KUKA KRL program: EPS_2_251455_MH10A_A_20251003045054.src

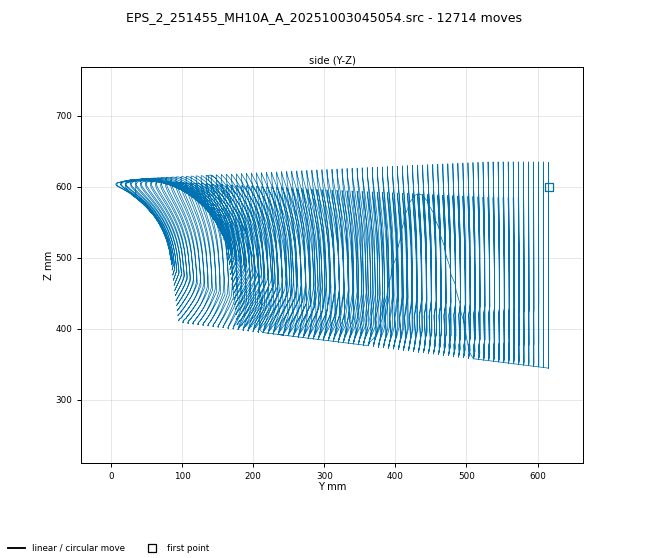
[picture p0: tool path of EPS_2_251455_MH10A_A_20251003045054.src, 12714 of 12716 moves have a stored position in this frame; points joined in program order, loops and branches not executed]
&ACCESS RVP
&REL 4
&COMMENT QRS 19112012
&PARAM EDITMASK = *
DEF PART()
EXT BAS (BAS_COMMAND :IN,REAL :IN )
INT I
BAS (#INITMOV,0 )

;KUKA QRS Post kuka4.cps  Date:22-06-2017 !

File_ID=2866

QRS_PRE_INIT()

;Init var - Until changes are made in qrs_pre_init
Outlet_Square_prg=0
Inlet_1_Square_prg=0
Inlet_2_Square_prg=0
Inlet_3_Square_prg=0
Inlet_4_Square_prg=0
Inlet_5_Square_prg=0

Outlet_1={X 0.000, Y 530.070, Z 534.500, B 0.000, E1 0.000 }
Inlet_1={X 0.000, Y 533.640, Z 484.500, B 0.000, E1 164.000 }
Outlet_1_type=201
Inlet_1_type=201
;QRS#1=Sidecore dimensions
;QRS#2=200-8" PVC SDR 35
;QRS#3=200-8" PVC SDR 35
;QRS#4=
;QRS#5=
;QRS#6=
;QRS#7=
;QRS#8=
;QRS#9=12-08 PSX
;QRS#10=12-08 PSX
;QRS#11=
;QRS#12=
;QRS#13=
;QRS#14=
;QRS#15=
;QRS#16=1220x127x914 3'
;QRS#17=EPS Height
;QRS#18=635
;QRS#19=*
;QRS#20= UPDATED VERSION 22-06-2017
;QRS#21=*
Outlet_Square=0100
Inlet_1_Square=0100
Inlet_2_Square=0
Inlet_3_Square=0
Inlet_4_Square=0
Inlet_5_Square=0
Mill_Square=1
Outlet_Square_Prg=204
Inlet_1_Square_prg=204

QRS_INIT()

$ADVANCE=5

; T1
PTP {E1 173.593,E2 173.593}
PTP {X 0,Y 615.507,A -85,B 0,C 180,E1 173.593,E2 173.593,E3 0,E4 0,E5 0,E6 0}
QRS_SPEED_INIT()
LIN {X 0,Y 615.507,Z 600,A -85,B 0,C 180,E1 173.593,E2 173.593,E3 0,E4 0,E5 0,E6 0} C_VEL
LIN {X 0,Y 615.507,Z 354.862,A -85,B 0,C 180,E1 173.593,E2 173.593} C_VEL
LIN {X 0,Y 615.507,Z 346.684,A -85,B 0,C 180,E1 173.593,E2 173.593} C_VEL
LIN {X 0,Y 615.492,Z 344.684,A -85,B 0,C 180,E1 173.407,E2 173.407} C_VEL
LIN {X 0,Y 615.497,Z 344.7,A -85,B 0,C 180,E1 170.801,E2 170.801} C_VEL
LIN {X 0,Y 615.474,Z 344.687,A -85,B 0,C 180,E1 168.139,E2 168.139} C_VEL
LIN {X 0,Y 615.493,Z 344.685,A -85,B 0,C 180,E1 165.451,E2 165.451} C_VEL
LIN {X 0,Y 615.497,Z 344.694,A -85,B 0,C 180,E1 162.729,E2 162.729} C_VEL
LIN {X 0,Y 615.479,Z 344.684,A -85,B 0,C 180,E1 159.967,E2 159.967} C_VEL
LIN {X 0,Y 615.489,Z 344.696,A -85,B 0,C 180,E1 157.155,E2 157.155} C_VEL
LIN {X 0,Y 615.478,Z 344.686,A -85,B 0,C 180,E1 154.283,E2 154.283} C_VEL
LIN {X 0,Y 615.495,Z 344.686,A -85,B 0,C 180,E1 151.546,E2 151.546} C_VEL
LIN {X 0,Y 615.494,Z 344.695,A -85,B 0,C 180,E1 148.911,E2 148.911} C_VEL
LIN {X 0,Y 615.484,Z 344.686,A -85,B 0,C 180,E1 146.464,E2 146.464} C_VEL
LIN {X 0,Y 615.477,Z 344.685,A -85,B 0,C 180,E1 144.166,E2 144.166} C_VEL
LIN {X 0,Y 615.484,Z 344.684,A -85,B 0,C 180,E1 141.931,E2 141.931} C_VEL
LIN {X 0,Y 615.492,Z 344.695,A -85,B 0,C 180,E1 139.393,E2 139.393} C_VEL
LIN {X 0,Y 615.498,Z 344.685,A -85,B 0,C 180,E1 136.756,E2 136.756} C_VEL
LIN {X 0,Y 615.483,Z 344.685,A -85,B 0,C 180,E1 133.996,E2 133.996} C_VEL
LIN {X 0,Y 615.493,Z 344.693,A -85,B 0,C 180,E1 131.094,E2 131.094} C_VEL
LIN {X 0,Y 615.492,Z 344.688,A -85,B 0,C 180,E1 128.903,E2 128.903} C_VEL
LIN {X 0,Y 615.479,Z 344.684,A -85,B 0,C 180,E1 126.424,E2 126.424} C_VEL
LIN {X 0,Y 615.484,Z 344.851,A -85,B 0,C 180,E1 123.96,E2 123.96} C_VEL
LIN {X 0,Y 615.482,Z 361.283,A -85,B 0,C 180,E1 121.084,E2 121.084} C_VEL
LIN {X 0,Y 615.497,Z 374.419,A -85,B 0,C 180,E1 118.808,E2 118.808} C_VEL
LIN {X 0,Y 615.481,Z 480.795,A -85,B 0,C 180,E1 117.545,E2 117.545} C_VEL
LIN {X 0,Y 615.478,Z 493.507,A -85,B 0,C 180,E1 117.269,E2 117.269} C_VEL
LIN {X 0,Y 615.495,Z 506.255,A -85,B 0,C 180,E1 116.855,E2 116.855} C_VEL
LIN {X 0,Y 615.483,Z 517.741,A -85,B 0,C 180,E1 116.352,E2 116.352} C_VEL
LIN {X 0,Y 615.495,Z 529.018,A -85,B 0,C 180,E1 115.715,E2 115.715} C_VEL
LIN {X 0,Y 615.499,Z 540.401,A -85,B 0,C 180,E1 114.9,E2 114.9} C_VEL
LIN {X 0,Y 615.499,Z 549.036,A -85,B 0,C 180,E1 114.14,E2 114.14} C_VEL
LIN {X 0,Y 615.497,Z 557.732,A -85,B 0,C 180,E1 113.199,E2 113.199} C_VEL
LIN {X 0,Y 615.496,Z 565.632,A -85,B 0,C 180,E1 112.136,E2 112.136} C_VEL
LIN {X 0,Y 615.497,Z 571.832,A -85,B 0,C 180,E1 111.08,E2 111.08} C_VEL
LIN {X 0,Y 615.496,Z 576.587,A -85,B 0,C 180,E1 110.032,E2 110.032} C_VEL
LIN {X 0,Y 615.495,Z 579.049,A -85,B 0,C 180,E1 109.337,E2 109.337} C_VEL
LIN {X 0,Y 615.496,Z 581.148,A -85,B 0,C 180,E1 108.605,E2 108.605} C_VEL
LIN {X 0,Y 615.498,Z 582.545,A -85,B 0,C 180,E1 107.956,E2 107.956} C_VEL
LIN {X 0,Y 615.496,Z 583.573,A -85,B 0,C 180,E1 107.27,E2 107.27} C_VEL
LIN {X 0,Y 615.496,Z 584.282,A -85,B 0,C 180,E1 106.432,E2 106.432} C_VEL
LIN {X 0,Y 615.497,Z 584.12,A -85,B 0,C 180,E1 105.225,E2 105.225} C_VEL
LIN {X 0,Y 615.499,Z 582.513,A -85,B 0,C 180,E1 103.935,E2 103.935} C_VEL
LIN {X 0,Y 615.495,Z 580.869,A -85,B 0,C 180,E1 103.201,E2 103.201} C_VEL
LIN {X 0,Y 615.496,Z 577.77,A -85,B 0,C 180,E1 102.195,E2 102.195} C_VEL
LIN {X 0,Y 615.497,Z 573.606,A -85,B 0,C 180,E1 101.193,E2 101.193} C_VEL
LIN {X 0,Y 615.496,Z 567.248,A -85,B 0,C 180,E1 100.028,E2 100.028} C_VEL
LIN {X 0,Y 615.496,Z 560.341,A -85,B 0,C 180,E1 99.033,E2 99.033} C_VEL
LIN {X 0,Y 615.499,Z 551.708,A -85,B 0,C 180,E1 98.04,E2 98.04} C_VEL
LIN {X 0,Y 615.497,Z 542.889,A -85,B 0,C 180,E1 97.215,E2 97.215} C_VEL
LIN {X 0,Y 615.496,Z 533.241,A -85,B 0,C 180,E1 96.474,E2 96.474} C_VEL
LIN {X 0,Y 615.492,Z 522.644,A -85,B 0,C 180,E1 95.816,E2 95.816} C_VEL
LIN {X 0,Y 615.496,Z 510.844,A -85,B 0,C 180,E1 95.241,E2 95.241} C_VEL
LIN {X 0,Y 615.486,Z 498.624,A -85,B 0,C 180,E1 94.79,E2 94.79} C_VEL
LIN {X 0,Y 615.477,Z 486.033,A -85,B 0,C 180,E1 94.461,E2 94.461} C_VEL
LIN {X 0,Y 615.482,Z 470.995,A -85,B 0,C 180,E1 94.236,E2 94.236} C_VEL
LIN {X 0,Y 615.491,Z 374.345,A -85,B 0,C 180,E1 93.089,E2 93.089} C_VEL
LIN {X 0,Y 615.484,Z 358.413,A -85,B 0,C 180,E1 90.327,E2 90.327} C_VEL
LIN {X 0,Y 615.488,Z 344.686,A -85,B 0,C 180,E1 87.914,E2 87.914} C_VEL
LIN {X 0,Y 615.478,Z 344.685,A -85,B 0,C 180,E1 85.415,E2 85.415} C_VEL
LIN {X 0,Y 615.495,Z 344.693,A -85,B 0,C 180,E1 82.785,E2 82.785} C_VEL
LIN {X 0,Y 615.495,Z 344.687,A -85,B 0,C 180,E1 80.138,E2 80.138} C_VEL
LIN {X 0,Y 615.478,Z 344.685,A -85,B 0,C 180,E1 77.47,E2 77.47} C_VEL
LIN {X 0,Y 615.494,Z 344.696,A -85,B 0,C 180,E1 74.775,E2 74.775} C_VEL
LIN {X 0,Y 615.495,Z 344.683,A -85,B 0,C 180,E1 72.044,E2 72.044} C_VEL
LIN {X 0,Y 615.488,Z 344.686,A -85,B 0,C 180,E1 69.27,E2 69.27} C_VEL
LIN {X 0,Y 615.492,Z 344.692,A -85,B 0,C 180,E1 66.444,E2 66.444} C_VEL
LIN {X 0,Y 615.494,Z 344.687,A -85,B 0,C 180,E1 64.285,E2 64.285} C_VEL
LIN {X 0,Y 615.477,Z 344.686,A -85,B 0,C 180,E1 61.553,E2 61.553} C_VEL
LIN {X 0,Y 615.496,Z 344.697,A -85,B 0,C 180,E1 58.914,E2 58.914} C_VEL
LIN {X 0,Y 615.483,Z 344.683,A -85,B 0,C 180,E1 55.979,E2 55.979} C_VEL
LIN {X 0,Y 615.493,Z 344.695,A -85,B 0,C 180,E1 53.063,E2 53.063} C_VEL
LIN {X 0,Y 615.495,Z 344.683,A -85,B 0,C 180,E1 50.252,E2 50.252} C_VEL
LIN {X 0,Y 615.476,Z 344.687,A -85,B 0,C 180,E1 47.647,E2 47.647} C_VEL
LIN {X 0,Y 615.493,Z 344.7,A -85,B 0,C 180,E1 44.933,E2 44.933} C_VEL
LIN {X 0,Y 615.486,Z 344.683,A -85,B 0,C 180,E1 42.082,E2 42.082} C_VEL
LIN {X 0,Y 615.477,Z 344.686,A -85,B 0,C 180,E1 39.751,E2 39.751} C_VEL
LIN {X 0,Y 615.492,Z 344.697,A -85,B 0,C 180,E1 36.939,E2 36.939} C_VEL
LIN {X 0,Y 615.481,Z 344.684,A -85,B 0,C 180,E1 34.023,E2 34.023} C_VEL
LIN {X 0,Y 615.479,Z 344.688,A -85,B 0,C 180,E1 31.686,E2 31.686} C_VEL
LIN {X 0,Y 615.489,Z 344.693,A -85,B 0,C 180,E1 29.407,E2 29.407} C_VEL
LIN {X 0,Y 615.494,Z 344.682,A -85,B 0,C 180,E1 26.444,E2 26.444} C_VEL
LIN {X 0,Y 615.485,Z 344.692,A -85,B 0,C 180,E1 23.557,E2 23.557} C_VEL
LIN {X 0,Y 615.484,Z 344.688,A -85,B 0,C 180,E1 20.731,E2 20.731} C_VEL
LIN {X 0,Y 615.477,Z 344.687,A -85,B 0,C 180,E1 17.958,E2 17.958} C_VEL
LIN {X 0,Y 615.491,Z 344.699,A -85,B 0,C 180,E1 15.226,E2 15.226} C_VEL
LIN {X 0,Y 615.485,Z 344.683,A -85,B 0,C 180,E1 12.53,E2 12.53} C_VEL
LIN {X 0,Y 615.477,Z 344.69,A -85,B 0,C 180,E1 9.863,E2 9.863} C_VEL
LIN {X 0,Y 615.483,Z 344.697,A -85,B 0,C 180,E1 7.216,E2 7.216} C_VEL
LIN {X 0,Y 615.492,Z 344.682,A -85,B 0,C 180,E1 4.585,E2 4.585} C_VEL
LIN {X 0,Y 615.477,Z 344.69,A -85,B 0,C 180,E1 1.963,E2 1.963} C_VEL
LIN {X 0,Y 615.486,Z 344.698,A -85,B 0,C 180,E1 -0.654,E2 -0.654} C_VEL
LIN {X 0,Y 615.485,Z 344.684,A -85,B 0,C 180,E1 -3.273,E2 -3.273} C_VEL
LIN {X 0,Y 615.476,Z 344.689,A -85,B 0,C 180,E1 -5.899,E2 -5.899} C_VEL
LIN {X 0,Y 615.486,Z 344.699,A -85,B 0,C 180,E1 -8.537,E2 -8.537} C_VEL
LIN {X 0,Y 615.483,Z 344.684,A -85,B 0,C 180,E1 -11.193,E2 -11.193} C_VEL
LIN {X 0,Y 615.48,Z 344.691,A -85,B 0,C 180,E1 -13.935,E2 -13.935} C_VEL
LIN {X 0,Y 615.482,Z 344.695,A -85,B 0,C 180,E1 -16.587,E2 -16.587} C_VEL
LIN {X 0,Y 615.486,Z 344.683,A -85,B 0,C 180,E1 -19.338,E2 -19.338} C_VEL
LIN {X 0,Y 615.488,Z 344.697,A -85,B 0,C 180,E1 -22.136,E2 -22.136} C_VEL
LIN {X 0,Y 615.476,Z 344.686,A -85,B 0,C 180,E1 -24.992,E2 -24.992} C_VEL
LIN {X 0,Y 615.482,Z 344.684,A -85,B 0,C 180,E1 -27.177,E2 -27.177} C_VEL
LIN {X 0,Y 615.483,Z 344.691,A -85,B 0,C 180,E1 -29.796,E2 -29.796} C_VEL
LIN {X 0,Y 615.489,Z 344.692,A -85,B 0,C 180,E1 -32.457,E2 -32.457} C_VEL
LIN {X 0,Y 615.477,Z 344.687,A -85,B 0,C 180,E1 -34.816,E2 -34.816} C_VEL
LIN {X 0,Y 615.489,Z 344.682,A -85,B 0,C 180,E1 -37.242,E2 -37.242} C_VEL
LIN {X 0,Y 615.497,Z 344.7,A -85,B 0,C 180,E1 -40.092,E2 -40.092} C_VEL
LIN {X 0,Y 615.493,Z 344.691,A -85,B 0,C 180,E1 -42.353,E2 -42.353} C_VEL
LIN {X 0,Y 615.481,Z 344.684,A -85,B 0,C 180,E1 -45.069,E2 -45.069} C_VEL
LIN {X 0,Y 615.494,Z 344.699,A -85,B 0,C 180,E1 -47.919,E2 -47.919} C_VEL
LIN {X 0,Y 615.495,Z 344.691,A -85,B 0,C 180,E1 -50.252,E2 -50.252} C_VEL
LIN {X 0,Y 615.483,Z 344.684,A -85,B 0,C 180,E1 -53.064,E2 -53.064} C_VEL
LIN {X 0,Y 615.497,Z 344.698,A -85,B 0,C 180,E1 -55.98,E2 -55.98} C_VEL
LIN {X 0,Y 615.487,Z 344.689,A -85,B 0,C 180,E1 -58.315,E2 -58.315} C_VEL
LIN {X 0,Y 615.477,Z 344.686,A -85,B 0,C 180,E1 -60.594,E2 -60.594} C_VEL
LIN {X 0,Y 615.486,Z 344.683,A -85,B 0,C 180,E1 -62.956,E2 -62.956} C_VEL
LIN {X 0,Y 615.491,Z 344.7,A -85,B 0,C 180,E1 -65.729,E2 -65.729} C_VEL
LIN {X 0,Y 615.487,Z 344.827,A -85,B 0,C 180,E1 -67.067,E2 -67.067} C_VEL
LIN {X 0,Y 615.484,Z 366.758,A -85,B 0,C 180,E1 -69.968,E2 -69.968} C_VEL
LIN {X 0,Y 615.478,Z 388,A -85,B 0,C 180,E1 -72.73,E2 -72.73} C_VEL
LIN {X 0,Y 615.479,Z 409.218,A -85,B 0,C 180,E1 -75.451,E2 -75.451} C_VEL
LIN {X 0,Y 615.497,Z 422.298,A -85,B 0,C 180,E1 -77.114,E2 -77.114} C_VEL
LIN {X 0,Y 615.479,Z 530.847,A -85,B 0,C 180,E1 -78.411,E2 -78.411} C_VEL
LIN {X 0,Y 615.478,Z 543.355,A -85,B 0,C 180,E1 -78.682,E2 -78.682} C_VEL
LIN {X 0,Y 615.491,Z 556.568,A -85,B 0,C 180,E1 -79.111,E2 -79.111} C_VEL
LIN {X 0,Y 615.478,Z 568.483,A -85,B 0,C 180,E1 -79.639,E2 -79.639} C_VEL
LIN {X 0,Y 615.487,Z 579.999,A -85,B 0,C 180,E1 -80.304,E2 -80.304} C_VEL
LIN {X 0,Y 615.499,Z 590.344,A -85,B 0,C 180,E1 -81.05,E2 -81.05} C_VEL
LIN {X 0,Y 615.497,Z 598.814,A -85,B 0,C 180,E1 -81.794,E2 -81.794} C_VEL
LIN {X 0,Y 615.498,Z 606.608,A -85,B 0,C 180,E1 -82.62,E2 -82.62} C_VEL
LIN {X 0,Y 615.496,Z 614.204,A -85,B 0,C 180,E1 -83.608,E2 -83.608} C_VEL
LIN {X 0,Y 615.498,Z 621.205,A -85,B 0,C 180,E1 -84.759,E2 -84.759} C_VEL
LIN {X 0,Y 615.493,Z 625.852,A -85,B 0,C 180,E1 -85.744,E2 -85.744} C_VEL
LIN {X 0,Y 615.495,Z 629.399,A -85,B 0,C 180,E1 -86.727,E2 -86.727} C_VEL
LIN {X 0,Y 615.497,Z 631.233,A -85,B 0,C 180,E1 -87.382,E2 -87.382} C_VEL
LIN {X 0,Y 615.497,Z 632.608,A -85,B 0,C 180,E1 -88.037,E2 -88.037} C_VEL
LIN {X 0,Y 615.496,Z 634.174,A -85,B 0,C 180,E1 -89.346,E2 -89.346} C_VEL
LIN {X 0,Y 615.494,Z 634.389,A -85,B 0,C 180,E1 -90,E2 -90} C_VEL
LIN {X 0,Y 615.496,Z 633.58,A -85,B 0,C 180,E1 -91.309,E2 -91.309} C_VEL
LIN {X 0,Y 615.497,Z 632.608,A -85,B 0,C 180,E1 -91.963,E2 -91.963} C_VEL
LIN {X 0,Y 615.497,Z 631.233,A -85,B 0,C 180,E1 -92.618,E2 -92.618} C_VEL
LIN {X 0,Y 615.496,Z 628.35,A -85,B 0,C 180,E1 -93.601,E2 -93.601} C_VEL
LIN {X 0,Y 615.498,Z 624.442,A -85,B 0,C 180,E1 -94.584,E2 -94.584} C_VEL
LIN {X 0,Y 615.499,Z 619.406,A -85,B 0,C 180,E1 -95.57,E2 -95.57} C_VEL
LIN {X 0,Y 615.497,Z 612.869,A -85,B 0,C 180,E1 -96.583,E2 -96.583} C_VEL
LIN {X 0,Y 615.497,Z 605.135,A -85,B 0,C 180,E1 -97.545,E2 -97.545} C_VEL
LIN {X 0,Y 615.498,Z 597.047,A -85,B 0,C 180,E1 -98.371,E2 -98.371} C_VEL
LIN {X 0,Y 615.499,Z 587.17,A -85,B 0,C 180,E1 -99.198,E2 -99.198} C_VEL
LIN {X 0,Y 615.488,Z 575.985,A -85,B 0,C 180,E1 -99.945,E2 -99.945} C_VEL
LIN {X 0,Y 615.481,Z 565.029,A -85,B 0,C 180,E1 -100.527,E2 -100.527} C_VEL
LIN {X 0,Y 615.49,Z 552.452,A -85,B 0,C 180,E1 -101.041,E2 -101.041} C_VEL
LIN {X 0,Y 615.477,Z 540.079,A -85,B 0,C 180,E1 -101.401,E2 -101.401} C_VEL
LIN {X 0,Y 615.481,Z 526.487,A -85,B 0,C 180,E1 -101.652,E2 -101.652} C_VEL
LIN {X 0,Y 615.497,Z 422.298,A -85,B 0,C 180,E1 -102.886,E2 -102.886} C_VEL
LIN {X 0,Y 615.485,Z 399.937,A -85,B 0,C 180,E1 -105.735,E2 -105.735} C_VEL
LIN {X 0,Y 615.481,Z 377.716,A -85,B 0,C 180,E1 -108.602,E2 -108.602} C_VEL
LIN {X 0,Y 615.478,Z 357.457,A -85,B 0,C 180,E1 -111.256,E2 -111.256} C_VEL
LIN {X 0,Y 615.486,Z 344.684,A -85,B 0,C 180,E1 -112.977,E2 -112.977} C_VEL
LIN {X 0,Y 615.489,Z 344.688,A -85,B 0,C 180,E1 -115.715,E2 -115.715} C_VEL
LIN {X 0,Y 615.49,Z 344.687,A -85,B 0,C 180,E1 -118.657,E2 -118.657} C_VEL
LIN {X 0,Y 615.482,Z 344.684,A -85,B 0,C 180,E1 -121.085,E2 -121.085} C_VEL
LIN {X 0,Y 615.498,Z 344.699,A -85,B 0,C 180,E1 -124.02,E2 -124.02} C_VEL
LIN {X 0,Y 615.483,Z 344.684,A -85,B 0,C 180,E1 -126.936,E2 -126.936} C_VEL
LIN {X 0,Y 615.495,Z 344.692,A -85,B 0,C 180,E1 -129.748,E2 -129.748} C_VEL
LIN {X 0,Y 615.484,Z 344.691,A -85,B 0,C 180,E1 -132.352,E2 -132.352} C_VEL
LIN {X 0,Y 615.479,Z 344.685,A -85,B 0,C 180,E1 -135.068,E2 -135.068} C_VEL
LIN {X 0,Y 615.497,Z 344.7,A -85,B 0,C 180,E1 -137.917,E2 -137.917} C_VEL
LIN {X 0,Y 615.483,Z 344.691,A -85,B 0,C 180,E1 -140.249,E2 -140.249} C_VEL
LIN {X 0,Y 615.478,Z 344.686,A -85,B 0,C 180,E1 -143.063,E2 -143.063} C_VEL
LIN {X 0,Y 615.487,Z 344.696,A -85,B 0,C 180,E1 -145.978,E2 -145.978} C_VEL
LIN {X 0,Y 615.481,Z 344.688,A -85,B 0,C 180,E1 -148.314,E2 -148.314} C_VEL
LIN {X 0,Y 615.487,Z 344.683,A -85,B 0,C 180,E1 -150.594,E2 -150.594} C_VEL
LIN {X 0,Y 615.493,Z 344.697,A -85,B 0,C 180,E1 -153.556,E2 -153.556} C_VEL
LIN {X 0,Y 615.485,Z 344.684,A -85,B 0,C 180,E1 -156.444,E2 -156.444} C_VEL
LIN {X 0,Y 615.48,Z 344.693,A -85,B 0,C 180,E1 -159.269,E2 -159.269} C_VEL
LIN {X 0,Y 615.477,Z 344.69,A -85,B 0,C 180,E1 -162.043,E2 -162.043} C_VEL
LIN {X 0,Y 615.487,Z 344.684,A -85,B 0,C 180,E1 -164.774,E2 -164.774} C_VEL
LIN {X 0,Y 615.488,Z 344.702,A -85,B 0,C 180,E1 -167.47,E2 -167.47} C_VEL
LIN {X 0,Y 615.477,Z 344.687,A -85,B 0,C 180,E1 -170.138,E2 -170.138} C_VEL
LIN {X 0,Y 615.486,Z 344.685,A -85,B 0,C 180,E1 -172.784,E2 -172.784} C_VEL
LIN {X 0,Y 615.5,Z 344.699,A -85,B 0,C 180,E1 -175.416,E2 -175.416} C_VEL
LIN {X 0,Y 615.477,Z 344.687,A -85,B 0,C 180,E1 -178.037,E2 -178.037} C_VEL
LIN {X 0,Y 615.488,Z 344.684,A -85,B 0,C 180,E1 -180.654,E2 -180.654} C_VEL
LIN {X 0,Y 615.493,Z 344.701,A -85,B 0,C 180,E1 -183.273,E2 -183.273} C_VEL
LIN {X 0,Y 615.476,Z 344.688,A -85,B 0,C 180,E1 -185.899,E2 -185.899} C_VEL
LIN {X 0,Y 615.492,Z 344.684,A -85,B 0,C 180,E1 -186.593,E2 -186.593} C_VEL
LIN {X 0,Y 614.818,Z 344.843,A -85,B 0,C 180,E1 -187.139,E2 -187.139} C_VEL
LIN {X 0,Y 611.987,Z 345.247,A -85,B 0,C 180,E1 -188.025,E2 -188.025} C_VEL
LIN {X 0,Y 609.594,Z 345.563,A -85,B 0,C 180,E1 -188.738,E2 -188.738} C_VEL
LIN {X 0,Y 608.554,Z 345.684,A -85,B 0,C 180,E1 -189.287,E2 -189.287} C_VEL
LIN {X 0,Y 608.462,Z 345.692,A -85,B 0,C 180,E1 -189.474,E2 -189.474} C_VEL
LIN {X 0,Y 608.453,Z 345.687,A -85,B 0,C 180,E1 -192,E2 -192} C_VEL
LIN {X 0,Y 608.48,Z 345.688,A -85,B 0,C 180,E1 -194.721,E2 -194.721} C_VEL
LIN {X 0,Y 608.456,Z 345.691,A -85,B 0,C 180,E1 -197.477,E2 -197.477} C_VEL
LIN {X 0,Y 608.461,Z 345.687,A -85,B 0,C 180,E1 -200.275,E2 -200.275} C_VEL
LIN {X 0,Y 608.486,Z 345.685,A -85,B 0,C 180,E1 -202.486,E2 -202.486} C_VEL
LIN {X 0,Y 608.453,Z 345.693,A -85,B 0,C 180,E1 -205.301,E2 -205.301} C_VEL
LIN {X 0,Y 608.449,Z 345.69,A -85,B 0,C 180,E1 -207.518,E2 -207.518} C_VEL
LIN {X 0,Y 608.46,Z 345.686,A -85,B 0,C 180,E1 -209.973,E2 -209.973} C_VEL
LIN {X 0,Y 608.467,Z 345.69,A -85,B 0,C 180,E1 -212.525,E2 -212.525} C_VEL
LIN {X 0,Y 608.444,Z 345.692,A -85,B 0,C 180,E1 -215.278,E2 -215.278} C_VEL
LIN {X 0,Y 608.468,Z 345.685,A -85,B 0,C 180,E1 -217.747,E2 -217.747} C_VEL
LIN {X 0,Y 608.452,Z 345.69,A -85,B 0,C 180,E1 -220.331,E2 -220.331} C_VEL
LIN {X 0,Y 608.484,Z 345.686,A -85,B 0,C 180,E1 -223.312,E2 -223.312} C_VEL
LIN {X 0,Y 608.469,Z 345.687,A -85,B 0,C 180,E1 -226.132,E2 -226.132} C_VEL
LIN {X 0,Y 608.463,Z 345.694,A -85,B 0,C 180,E1 -228.825,E2 -228.825} C_VEL
LIN {X 0,Y 608.471,Z 345.686,A -85,B 0,C 180,E1 -231.413,E2 -231.413} C_VEL
LIN {X 0,Y 608.478,Z 345.686,A -85,B 0,C 180,E1 -233.951,E2 -233.951} C_VEL
LIN {X 0,Y 608.477,Z 345.815,A -85,B 0,C 180,E1 -235.982,E2 -235.982} C_VEL
LIN {X 0,Y 608.478,Z 361.372,A -85,B 0,C 180,E1 -238.729,E2 -238.729} C_VEL
LIN {X 0,Y 608.468,Z 374.62,A -85,B 0,C 180,E1 -241.04,E2 -241.04} C_VEL
LIN {X 0,Y 608.552,Z 481.725,A -85,B 0,C 180,E1 -242.336,E2 -242.336} C_VEL
LIN {X 0,Y 608.522,Z 495.158,A -85,B 0,C 180,E1 -242.643,E2 -242.643} C_VEL
LIN {X 0,Y 608.536,Z 507.968,A -85,B 0,C 180,E1 -243.079,E2 -243.079} C_VEL
LIN {X 0,Y 608.509,Z 519.292,A -85,B 0,C 180,E1 -243.599,E2 -243.599} C_VEL
LIN {X 0,Y 608.5,Z 530.782,A -85,B 0,C 180,E1 -244.275,E2 -244.275} C_VEL
LIN {X 0,Y 608.484,Z 541.548,A -85,B 0,C 180,E1 -245.067,E2 -245.067} C_VEL
LIN {X 0,Y 608.466,Z 550.208,A -85,B 0,C 180,E1 -245.851,E2 -245.851} C_VEL
LIN {X 0,Y 608.471,Z 559.405,A -85,B 0,C 180,E1 -246.877,E2 -246.877} C_VEL
LIN {X 0,Y 608.455,Z 567.1,A -85,B 0,C 180,E1 -247.952,E2 -247.952} C_VEL
LIN {X 0,Y 608.434,Z 573.088,A -85,B 0,C 180,E1 -249.018,E2 -249.018} C_VEL
LIN {X 0,Y 608.435,Z 577.702,A -85,B 0,C 180,E1 -250.078,E2 -250.078} C_VEL
LIN {X 0,Y 608.43,Z 581.545,A -85,B 0,C 180,E1 -251.297,E2 -251.297} C_VEL
LIN {X 0,Y 608.421,Z 583.95,A -85,B 0,C 180,E1 -252.523,E2 -252.523} C_VEL
LIN {X 0,Y 608.423,Z 584.856,A -85,B 0,C 180,E1 -253.487,E2 -253.487} C_VEL
LIN {X 0,Y 608.42,Z 584.862,A -85,B 0,C 180,E1 -254.593,E2 -254.593} C_VEL
LIN {X 0,Y 608.418,Z 584.29,A -85,B 0,C 180,E1 -255.278,E2 -255.278} C_VEL
LIN {X 0,Y 608.446,Z 583.262,A -85,B 0,C 180,E1 -255.994,E2 -255.994} C_VEL
LIN {X 0,Y 608.438,Z 581.93,A -85,B 0,C 180,E1 -256.643,E2 -256.643} C_VEL
LIN {X 0,Y 608.433,Z 578.981,A -85,B 0,C 180,E1 -257.661,E2 -257.661} C_VEL
LIN {X 0,Y 608.43,Z 574.981,A -85,B 0,C 180,E1 -258.676,E2 -258.676} C_VEL
LIN {X 0,Y 608.444,Z 568.822,A -85,B 0,C 180,E1 -259.855,E2 -259.855} C_VEL
LIN {X 0,Y 608.47,Z 562.103,A -85,B 0,C 180,E1 -260.862,E2 -260.862} C_VEL
LIN {X 0,Y 608.464,Z 553.803,A -85,B 0,C 180,E1 -261.866,E2 -261.866} C_VEL
LIN {X 0,Y 608.478,Z 545.303,A -85,B 0,C 180,E1 -262.701,E2 -262.701} C_VEL
LIN {X 0,Y 608.481,Z 534.872,A -85,B 0,C 180,E1 -263.534,E2 -263.534} C_VEL
LIN {X 0,Y 608.513,Z 524.576,A -85,B 0,C 180,E1 -264.2,E2 -264.2} C_VEL
LIN {X 0,Y 608.53,Z 513.328,A -85,B 0,C 180,E1 -264.782,E2 -264.782} C_VEL
LIN {X 0,Y 608.527,Z 501.849,A -85,B 0,C 180,E1 -265.239,E2 -265.239} C_VEL
LIN {X 0,Y 608.539,Z 488.732,A -85,B 0,C 180,E1 -265.612,E2 -265.612} C_VEL
LIN {X 0,Y 608.544,Z 476.006,A -85,B 0,C 180,E1 -265.84,E2 -265.84} C_VEL
LIN {X 0,Y 608.485,Z 374.794,A -85,B 0,C 180,E1 -267.041,E2 -267.041} C_VEL
LIN {X 0,Y 608.46,Z 359.621,A -85,B 0,C 180,E1 -269.669,E2 -269.669} C_VEL
LIN {X 0,Y 608.466,Z 345.688,A -85,B 0,C 180,E1 -272.151,E2 -272.151} C_VEL
LIN {X 0,Y 608.448,Z 345.688,A -85,B 0,C 180,E1 -274.638,E2 -274.638} C_VEL
LIN {X 0,Y 608.472,Z 345.693,A -85,B 0,C 180,E1 -277.299,E2 -277.299} C_VEL
LIN {X 0,Y 608.462,Z 345.688,A -85,B 0,C 180,E1 -279.977,E2 -279.977} C_VEL
LIN {X 0,Y 608.472,Z 345.686,A -85,B 0,C 180,E1 -282.677,E2 -282.677} C_VEL
LIN {X 0,Y 608.478,Z 345.694,A -85,B 0,C 180,E1 -285.405,E2 -285.405} C_VEL
LIN {X 0,Y 608.454,Z 345.687,A -85,B 0,C 180,E1 -288.171,E2 -288.171} C_VEL
LIN {X 0,Y 608.46,Z 345.692,A -85,B 0,C 180,E1 -290.981,E2 -290.981} C_VEL
LIN {X 0,Y 608.469,Z 345.687,A -85,B 0,C 180,E1 -293.844,E2 -293.844} C_VEL
LIN {X 0,Y 608.447,Z 345.688,A -85,B 0,C 180,E1 -296.035,E2 -296.035} C_VEL
LIN {X 0,Y 608.47,Z 345.687,A -85,B 0,C 180,E1 -298.618,E2 -298.618} C_VEL
LIN {X 0,Y 608.481,Z 345.692,A -85,B 0,C 180,E1 -301.315,E2 -301.315} C_VEL
LIN {X 0,Y 608.474,Z 345.686,A -85,B 0,C 180,E1 -303.734,E2 -303.734} C_VEL
LIN {X 0,Y 608.476,Z 345.684,A -85,B 0,C 180,E1 -306.089,E2 -306.089} C_VEL
LIN {X 0,Y 608.473,Z 345.687,A -85,B 0,C 180,E1 -308.587,E2 -308.587} C_VEL
LIN {X 0,Y 608.464,Z 345.692,A -85,B 0,C 180,E1 -311.342,E2 -311.342} C_VEL
LIN {X 0,Y 608.45,Z 345.688,A -85,B 0,C 180,E1 -314.263,E2 -314.263} C_VEL
LIN {X 0,Y 608.462,Z 345.697,A -85,B 0,C 180,E1 -317.04,E2 -317.04} C_VEL
LIN {X 0,Y 608.453,Z 345.688,A -85,B 0,C 180,E1 -319.696,E2 -319.696} C_VEL
LIN {X 0,Y 608.469,Z 345.686,A -85,B 0,C 180,E1 -322.253,E2 -322.253} C_VEL
LIN {X 0,Y 608.474,Z 345.692,A -85,B 0,C 180,E1 -325.089,E2 -325.089} C_VEL
LIN {X 0,Y 608.469,Z 345.685,A -85,B 0,C 180,E1 -327.905,E2 -327.905} C_VEL
LIN {X 0,Y 608.462,Z 345.688,A -85,B 0,C 180,E1 -330.22,E2 -330.22} C_VEL
LIN {X 0,Y 608.482,Z 345.694,A -85,B 0,C 180,E1 -332.789,E2 -332.789} C_VEL
LIN {X 0,Y 608.454,Z 345.689,A -85,B 0,C 180,E1 -335.429,E2 -335.429} C_VEL
LIN {X 0,Y 608.471,Z 345.688,A -85,B 0,C 180,E1 -338.308,E2 -338.308} C_VEL
LIN {X 0,Y 608.467,Z 345.688,A -85,B 0,C 180,E1 -341.281,E2 -341.281} C_VEL
LIN {X 0,Y 608.456,Z 345.687,A -85,B 0,C 180,E1 -343.906,E2 -343.906} C_VEL
LIN {X 0,Y 608.465,Z 345.696,A -85,B 0,C 180,E1 -346.643,E2 -346.643} C_VEL
LIN {X 0,Y 608.466,Z 345.686,A -85,B 0,C 180,E1 -349.35,E2 -349.35} C_VEL
LIN {X 0,Y 608.47,Z 345.687,A -85,B 0,C 180,E1 -352.033,E2 -352.033} C_VEL
LIN {X 0,Y 608.465,Z 345.694,A -85,B 0,C 180,E1 -354.698,E2 -354.698} C_VEL
LIN {X 0,Y 608.479,Z 345.684,A -85,B 0,C 180,E1 -357.352,E2 -357.352} C_VEL
LIN {X 0,Y 608.468,Z 345.688,A -85,B 0,C 180,E1 -360,E2 -360} C_VEL
LIN {X 0,Y 608.48,Z 345.692,A -85,B 0,C 180,E1 -362.648,E2 -362.648} C_VEL
LIN {X 0,Y 608.462,Z 345.686,A -85,B 0,C 180,E1 -365.302,E2 -365.302} C_VEL
LIN {X 0,Y 608.47,Z 345.688,A -85,B 0,C 180,E1 -367.967,E2 -367.967} C_VEL
LIN {X 0,Y 608.465,Z 345.692,A -85,B 0,C 180,E1 -370.65,E2 -370.65} C_VEL
LIN {X 0,Y 608.46,Z 345.686,A -85,B 0,C 180,E1 -373.356,E2 -373.356} C_VEL
LIN {X 0,Y 608.458,Z 345.693,A -85,B 0,C 180,E1 -376.094,E2 -376.094} C_VEL
LIN {X 0,Y 608.45,Z 345.69,A -85,B 0,C 180,E1 -378.87,E2 -378.87} C_VEL
LIN {X 0,Y 608.473,Z 345.687,A -85,B 0,C 180,E1 -381.691,E2 -381.691} C_VEL
LIN {X 0,Y 608.451,Z 345.693,A -85,B 0,C 180,E1 -384.571,E2 -384.571} C_VEL
LIN {X 0,Y 608.473,Z 345.685,A -85,B 0,C 180,E1 -387.209,E2 -387.209} C_VEL
LIN {X 0,Y 608.468,Z 345.692,A -85,B 0,C 180,E1 -389.974,E2 -389.974} C_VEL
LIN {X 0,Y 608.462,Z 345.691,A -85,B 0,C 180,E1 -392.525,E2 -392.525} C_VEL
LIN {X 0,Y 608.439,Z 345.689,A -85,B 0,C 180,E1 -395.278,E2 -395.278} C_VEL
LIN {X 0,Y 608.472,Z 345.689,A -85,B 0,C 180,E1 -397.746,E2 -397.746} C_VEL
LIN {X 0,Y 608.476,Z 345.69,A -85,B 0,C 180,E1 -400.333,E2 -400.333} C_VEL
LIN {X 0,Y 608.483,Z 345.684,A -85,B 0,C 180,E1 -403.312,E2 -403.312} C_VEL
LIN {X 0,Y 608.472,Z 345.693,A -85,B 0,C 180,E1 -406.132,E2 -406.132} C_VEL
LIN {X 0,Y 608.45,Z 345.688,A -85,B 0,C 180,E1 -408.824,E2 -408.824} C_VEL
LIN {X 0,Y 608.471,Z 345.687,A -85,B 0,C 180,E1 -411.413,E2 -411.413} C_VEL
LIN {X 0,Y 608.478,Z 345.695,A -85,B 0,C 180,E1 -413.951,E2 -413.951} C_VEL
LIN {X 0,Y 608.464,Z 345.689,A -85,B 0,C 180,E1 -416.33,E2 -416.33} C_VEL
LIN {X 0,Y 608.476,Z 345.685,A -85,B 0,C 180,E1 -418.728,E2 -418.728} C_VEL
LIN {X 0,Y 608.477,Z 345.688,A -85,B 0,C 180,E1 -421.38,E2 -421.38} C_VEL
LIN {X 0,Y 608.471,Z 345.688,A -85,B 0,C 180,E1 -424.28,E2 -424.28} C_VEL
LIN {X 0,Y 608.479,Z 345.824,A -85,B 0,C 180,E1 -426.923,E2 -426.923} C_VEL
LIN {X 0,Y 608.582,Z 361.447,A -85,B 0,C 180,E1 -429.024,E2 -429.024} C_VEL
LIN {X 0,Y 608.518,Z 382.72,A -85,B 0,C 180,E1 -431.831,E2 -431.831} C_VEL
LIN {X 0,Y 608.492,Z 402.663,A -85,B 0,C 180,E1 -434.423,E2 -434.423} C_VEL
LIN {X 0,Y 608.503,Z 422.524,A -85,B 0,C 180,E1 -436.974,E2 -436.974} C_VEL
LIN {X 0,Y 608.538,Z 530.962,A -85,B 0,C 180,E1 -438.277,E2 -438.277} C_VEL
LIN {X 0,Y 608.514,Z 544.226,A -85,B 0,C 180,E1 -438.572,E2 -438.572} C_VEL
LIN {X 0,Y 608.517,Z 556.598,A -85,B 0,C 180,E1 -438.981,E2 -438.981} C_VEL
LIN {X 0,Y 608.498,Z 568.639,A -85,B 0,C 180,E1 -439.519,E2 -439.519} C_VEL
LIN {X 0,Y 608.48,Z 580.201,A -85,B 0,C 180,E1 -440.191,E2 -440.191} C_VEL
LIN {X 0,Y 608.485,Z 590.596,A -85,B 0,C 180,E1 -440.946,E2 -440.946} C_VEL
LIN {X 0,Y 608.475,Z 599.114,A -85,B 0,C 180,E1 -441.699,E2 -441.699} C_VEL
LIN {X 0,Y 608.471,Z 606.962,A -85,B 0,C 180,E1 -442.534,E2 -442.534} C_VEL
LIN {X 0,Y 608.46,Z 614.287,A -85,B 0,C 180,E1 -443.485,E2 -443.485} C_VEL
LIN {X 0,Y 608.45,Z 619.867,A -85,B 0,C 180,E1 -444.366,E2 -444.366} C_VEL
LIN {X 0,Y 608.432,Z 624.951,A -85,B 0,C 180,E1 -445.362,E2 -445.362} C_VEL
LIN {X 0,Y 608.449,Z 628.896,A -85,B 0,C 180,E1 -446.358,E2 -446.358} C_VEL
LIN {X 0,Y 608.425,Z 631.809,A -85,B 0,C 180,E1 -447.352,E2 -447.352} C_VEL
LIN {X 0,Y 608.442,Z 633.201,A -85,B 0,C 180,E1 -448.014,E2 -448.014} C_VEL
LIN {X 0,Y 608.438,Z 634.783,A -85,B 0,C 180,E1 -449.338,E2 -449.338} C_VEL
LIN {X 0,Y 608.434,Z 635,A -85,B 0,C 180,E1 -450,E2 -450} C_VEL
LIN {X 0,Y 608.448,Z 634.184,A -85,B 0,C 180,E1 -451.324,E2 -451.324} C_VEL
LIN {X 0,Y 608.442,Z 633.201,A -85,B 0,C 180,E1 -451.986,E2 -451.986} C_VEL
LIN {X 0,Y 608.425,Z 631.809,A -85,B 0,C 180,E1 -452.648,E2 -452.648} C_VEL
LIN {X 0,Y 608.449,Z 628.896,A -85,B 0,C 180,E1 -453.642,E2 -453.642} C_VEL
LIN {X 0,Y 608.432,Z 624.95,A -85,B 0,C 180,E1 -454.638,E2 -454.638} C_VEL
LIN {X 0,Y 608.437,Z 618.877,A -85,B 0,C 180,E1 -455.801,E2 -455.801} C_VEL
LIN {X 0,Y 608.462,Z 612.236,A -85,B 0,C 180,E1 -456.799,E2 -456.799} C_VEL
LIN {X 0,Y 608.455,Z 603.991,A -85,B 0,C 180,E1 -457.8,E2 -457.8} C_VEL
LIN {X 0,Y 608.472,Z 595.538,A -85,B 0,C 180,E1 -458.636,E2 -458.636} C_VEL
LIN {X 0,Y 608.471,Z 585.094,A -85,B 0,C 180,E1 -459.473,E2 -459.473} C_VEL
LIN {X 0,Y 608.494,Z 574.76,A -85,B 0,C 180,E1 -460.144,E2 -460.144} C_VEL
LIN {X 0,Y 608.521,Z 563.255,A -85,B 0,C 180,E1 -460.74,E2 -460.74} C_VEL
LIN {X 0,Y 608.531,Z 550.887,A -85,B 0,C 180,E1 -461.225,E2 -461.225} C_VEL
LIN {X 0,Y 608.537,Z 537.45,A -85,B 0,C 180,E1 -461.597,E2 -461.597} C_VEL
LIN {X 0,Y 608.546,Z 525.105,A -85,B 0,C 180,E1 -461.808,E2 -461.808} C_VEL
LIN {X 0,Y 608.493,Z 422.441,A -85,B 0,C 180,E1 -463.037,E2 -463.037} C_VEL
LIN {X 0,Y 608.494,Z 400.004,A -85,B 0,C 180,E1 -465.92,E2 -465.92} C_VEL
LIN {X 0,Y 608.54,Z 378.405,A -85,B 0,C 180,E1 -468.735,E2 -468.735} C_VEL
LIN {X 0,Y 608.563,Z 357.458,A -85,B 0,C 180,E1 -471.51,E2 -471.51} C_VEL
LIN {X 0,Y 608.468,Z 345.687,A -85,B 0,C 180,E1 -473.1,E2 -473.1} C_VEL
LIN {X 0,Y 608.471,Z 345.688,A -85,B 0,C 180,E1 -475.72,E2 -475.72} C_VEL
LIN {X 0,Y 608.476,Z 345.688,A -85,B 0,C 180,E1 -478.62,E2 -478.62} C_VEL
LIN {X 0,Y 608.475,Z 345.685,A -85,B 0,C 180,E1 -481.315,E2 -481.315} C_VEL
LIN {X 0,Y 608.473,Z 345.69,A -85,B 0,C 180,E1 -483.735,E2 -483.735} C_VEL
LIN {X 0,Y 608.477,Z 345.695,A -85,B 0,C 180,E1 -486.089,E2 -486.089} C_VEL
LIN {X 0,Y 608.471,Z 345.687,A -85,B 0,C 180,E1 -488.587,E2 -488.587} C_VEL
LIN {X 0,Y 608.457,Z 345.688,A -85,B 0,C 180,E1 -491.341,E2 -491.341} C_VEL
LIN {X 0,Y 608.457,Z 345.692,A -85,B 0,C 180,E1 -494.264,E2 -494.264} C_VEL
LIN {X 0,Y 608.453,Z 345.687,A -85,B 0,C 180,E1 -497.04,E2 -497.04} C_VEL
LIN {X 0,Y 608.455,Z 345.695,A -85,B 0,C 180,E1 -499.697,E2 -499.697} C_VEL
LIN {X 0,Y 608.471,Z 345.689,A -85,B 0,C 180,E1 -502.254,E2 -502.254} C_VEL
LIN {X 0,Y 608.469,Z 345.686,A -85,B 0,C 180,E1 -505.09,E2 -505.09} C_VEL
LIN {X 0,Y 608.47,Z 345.693,A -85,B 0,C 180,E1 -507.906,E2 -507.906} C_VEL
LIN {X 0,Y 608.464,Z 345.689,A -85,B 0,C 180,E1 -510.22,E2 -510.22} C_VEL
LIN {X 0,Y 608.475,Z 345.685,A -85,B 0,C 180,E1 -512.791,E2 -512.791} C_VEL
LIN {X 0,Y 608.449,Z 345.694,A -85,B 0,C 180,E1 -515.429,E2 -515.429} C_VEL
LIN {X 0,Y 608.471,Z 345.686,A -85,B 0,C 180,E1 -518.309,E2 -518.309} C_VEL
LIN {X 0,Y 608.466,Z 345.691,A -85,B 0,C 180,E1 -521.281,E2 -521.281} C_VEL
LIN {X 0,Y 608.456,Z 345.691,A -85,B 0,C 180,E1 -523.906,E2 -523.906} C_VEL
LIN {X 0,Y 608.46,Z 345.686,A -85,B 0,C 180,E1 -526.644,E2 -526.644} C_VEL
LIN {X 0,Y 608.466,Z 345.694,A -85,B 0,C 180,E1 -529.35,E2 -529.35} C_VEL
LIN {X 0,Y 608.47,Z 345.687,A -85,B 0,C 180,E1 -532.033,E2 -532.033} C_VEL
LIN {X 0,Y 608.464,Z 345.687,A -85,B 0,C 180,E1 -534.698,E2 -534.698} C_VEL
LIN {X 0,Y 608.484,Z 345.694,A -85,B 0,C 180,E1 -537.352,E2 -537.352} C_VEL
LIN {X 0,Y 608.468,Z 345.687,A -85,B 0,C 180,E1 -540,E2 -540} C_VEL
LIN {X 0,Y 608.482,Z 345.685,A -85,B 0,C 180,E1 -542.648,E2 -542.648} C_VEL
LIN {X 0,Y 608.473,Z 345.695,A -85,B 0,C 180,E1 -545.302,E2 -545.302} C_VEL
LIN {X 0,Y 608.47,Z 345.686,A -85,B 0,C 180,E1 -547.967,E2 -547.967} C_VEL
LIN {X 0,Y 608.462,Z 345.692,A -85,B 0,C 180,E1 -549.474,E2 -549.474} C_VEL
LIN {X 0,Y 607.774,Z 345.774,A -85,B 0,C 180,E1 -550.026,E2 -550.026} C_VEL
LIN {X 0,Y 604.913,Z 346.134,A -85,B 0,C 180,E1 -550.923,E2 -550.923} C_VEL
LIN {X 0,Y 602.511,Z 346.43,A -85,B 0,C 180,E1 -551.645,E2 -551.645} C_VEL
LIN {X 0,Y 601.487,Z 346.555,A -85,B 0,C 180,E1 -552.201,E2 -552.201} C_VEL
LIN {X 0,Y 601.406,Z 346.565,A -85,B 0,C 180,E1 -552.39,E2 -552.39} C_VEL
LIN {X 0,Y 601.433,Z 346.568,A -85,B 0,C 180,E1 -554.897,E2 -554.897} C_VEL
LIN {X 0,Y 601.398,Z 346.568,A -85,B 0,C 180,E1 -557.689,E2 -557.689} C_VEL
LIN {X 0,Y 601.431,Z 346.564,A -85,B 0,C 180,E1 -560.522,E2 -560.522} C_VEL
LIN {X 0,Y 601.418,Z 346.568,A -85,B 0,C 180,E1 -563.411,E2 -563.411} C_VEL
LIN {X 0,Y 601.406,Z 346.567,A -85,B 0,C 180,E1 -566.364,E2 -566.364} C_VEL
LIN {X 0,Y 601.442,Z 346.569,A -85,B 0,C 180,E1 -568.792,E2 -568.792} C_VEL
LIN {X 0,Y 601.413,Z 346.565,A -85,B 0,C 180,E1 -571.727,E2 -571.727} C_VEL
LIN {X 0,Y 601.428,Z 346.563,A -85,B 0,C 180,E1 -574.119,E2 -574.119} C_VEL
LIN {X 0,Y 601.413,Z 346.57,A -85,B 0,C 180,E1 -576.583,E2 -576.583} C_VEL
LIN {X 0,Y 601.436,Z 346.562,A -85,B 0,C 180,E1 -579.537,E2 -579.537} C_VEL
LIN {X 0,Y 601.438,Z 346.569,A -85,B 0,C 180,E1 -582.595,E2 -582.595} C_VEL
LIN {X 0,Y 601.423,Z 346.564,A -85,B 0,C 180,E1 -585.483,E2 -585.483} C_VEL
LIN {X 0,Y 601.427,Z 346.568,A -85,B 0,C 180,E1 -588.407,E2 -588.407} C_VEL
LIN {X 0,Y 601.439,Z 346.568,A -85,B 0,C 180,E1 -590.877,E2 -590.877} C_VEL
LIN {X 0,Y 601.444,Z 346.561,A -85,B 0,C 180,E1 -593.735,E2 -593.735} C_VEL
LIN {X 0,Y 601.42,Z 346.646,A -85,B 0,C 180,E1 -595.912,E2 -595.912} C_VEL
LIN {X 0,Y 601.443,Z 361.359,A -85,B 0,C 180,E1 -598.543,E2 -598.543} C_VEL
LIN {X 0,Y 601.412,Z 374.66,A -85,B 0,C 180,E1 -600.891,E2 -600.891} C_VEL
LIN {X 0,Y 601.684,Z 380.406,A -85,B 0,C 180,E1 -600.966,E2 -600.966} C_VEL
LIN {X 0,Y 601.594,Z 481.501,A -85,B 0,C 180,E1 -602.195,E2 -602.195} C_VEL
LIN {X 0,Y 601.551,Z 495.079,A -85,B 0,C 180,E1 -602.507,E2 -602.507} C_VEL
LIN {X 0,Y 601.564,Z 507.771,A -85,B 0,C 180,E1 -602.942,E2 -602.942} C_VEL
LIN {X 0,Y 601.499,Z 518.891,A -85,B 0,C 180,E1 -603.455,E2 -603.455} C_VEL
LIN {X 0,Y 601.465,Z 530.246,A -85,B 0,C 180,E1 -604.124,E2 -604.124} C_VEL
LIN {X 0,Y 601.465,Z 541.295,A -85,B 0,C 180,E1 -604.94,E2 -604.94} C_VEL
LIN {X 0,Y 601.4,Z 551.203,A -85,B 0,C 180,E1 -605.858,E2 -605.858} C_VEL
LIN {X 0,Y 601.386,Z 559.233,A -85,B 0,C 180,E1 -606.771,E2 -606.771} C_VEL
LIN {X 0,Y 601.392,Z 566.085,A -85,B 0,C 180,E1 -607.723,E2 -607.723} C_VEL
LIN {X 0,Y 601.344,Z 572.104,A -85,B 0,C 180,E1 -608.759,E2 -608.759} C_VEL
LIN {X 0,Y 601.342,Z 576.969,A -85,B 0,C 180,E1 -609.833,E2 -609.833} C_VEL
LIN {X 0,Y 601.332,Z 580.578,A -85,B 0,C 180,E1 -610.899,E2 -610.899} C_VEL
LIN {X 0,Y 601.325,Z 582.338,A -85,B 0,C 180,E1 -611.606,E2 -611.606} C_VEL
LIN {X 0,Y 601.314,Z 583.652,A -85,B 0,C 180,E1 -612.31,E2 -612.31} C_VEL
LIN {X 0,Y 601.322,Z 584.81,A -85,B 0,C 180,E1 -613.414,E2 -613.414} C_VEL
LIN {X 0,Y 601.327,Z 584.922,A -85,B 0,C 180,E1 -614.407,E2 -614.407} C_VEL
LIN {X 0,Y 601.315,Z 584.508,A -85,B 0,C 180,E1 -615.101,E2 -615.101} C_VEL
LIN {X 0,Y 601.353,Z 583.395,A -85,B 0,C 180,E1 -615.937,E2 -615.937} C_VEL
LIN {X 0,Y 601.328,Z 580.634,A -85,B 0,C 180,E1 -617.17,E2 -617.17} C_VEL
LIN {X 0,Y 601.351,Z 577.188,A -85,B 0,C 180,E1 -618.199,E2 -618.199} C_VEL
LIN {X 0,Y 601.34,Z 572.649,A -85,B 0,C 180,E1 -619.223,E2 -619.223} C_VEL
LIN {X 0,Y 601.377,Z 565.774,A -85,B 0,C 180,E1 -620.414,E2 -620.414} C_VEL
LIN {X 0,Y 601.407,Z 558.324,A -85,B 0,C 180,E1 -621.431,E2 -621.431} C_VEL
LIN {X 0,Y 601.397,Z 550.774,A -85,B 0,C 180,E1 -622.277,E2 -622.277} C_VEL
LIN {X 0,Y 601.452,Z 541.647,A -85,B 0,C 180,E1 -623.121,E2 -623.121} C_VEL
LIN {X 0,Y 601.485,Z 530.28,A -85,B 0,C 180,E1 -623.964,E2 -623.964} C_VEL
LIN {X 0,Y 601.5,Z 518.868,A -85,B 0,C 180,E1 -624.637,E2 -624.637} C_VEL
LIN {X 0,Y 601.573,Z 506.846,A -85,B 0,C 180,E1 -625.183,E2 -625.183} C_VEL
LIN {X 0,Y 601.554,Z 493.636,A -85,B 0,C 180,E1 -625.624,E2 -625.624} C_VEL
LIN {X 0,Y 601.591,Z 480.258,A -85,B 0,C 180,E1 -625.918,E2 -625.918} C_VEL
LIN {X 0,Y 601.542,Z 375.529,A -85,B 0,C 180,E1 -627.185,E2 -627.185} C_VEL
LIN {X 0,Y 601.413,Z 374.442,A -85,B 0,C 180,E1 -627.237,E2 -627.237} C_VEL
LIN {X 0,Y 601.451,Z 358.811,A -85,B 0,C 180,E1 -630,E2 -630} C_VEL
LIN {X 0,Y 601.424,Z 346.566,A -85,B 0,C 180,E1 -632.218,E2 -632.218} C_VEL
LIN {X 0,Y 601.419,Z 346.564,A -85,B 0,C 180,E1 -634.692,E2 -634.692} C_VEL
LIN {X 0,Y 601.449,Z 346.57,A -85,B 0,C 180,E1 -637.385,E2 -637.385} C_VEL
LIN {X 0,Y 601.438,Z 346.562,A -85,B 0,C 180,E1 -640.095,E2 -640.095} C_VEL
LIN {X 0,Y 601.42,Z 346.565,A -85,B 0,C 180,E1 -642.828,E2 -642.828} C_VEL
LIN {X 0,Y 601.419,Z 346.57,A -85,B 0,C 180,E1 -645.591,E2 -645.591} C_VEL
LIN {X 0,Y 601.424,Z 346.563,A -85,B 0,C 180,E1 -648.391,E2 -648.391} C_VEL
LIN {X 0,Y 601.412,Z 346.574,A -85,B 0,C 180,E1 -651.239,E2 -651.239} C_VEL
LIN {X 0,Y 601.456,Z 346.559,A -85,B 0,C 180,E1 -654.14,E2 -654.14} C_VEL
LIN {X 0,Y 601.455,Z 346.568,A -85,B 0,C 180,E1 -657.11,E2 -657.11} C_VEL
LIN {X 0,Y 601.426,Z 346.57,A -85,B 0,C 180,E1 -659.392,E2 -659.392} C_VEL
LIN {X 0,Y 601.414,Z 346.566,A -85,B 0,C 180,E1 -661.725,E2 -661.725} C_VEL
LIN {X 0,Y 601.431,Z 346.562,A -85,B 0,C 180,E1 -664.117,E2 -664.117} C_VEL
LIN {X 0,Y 601.416,Z 346.566,A -85,B 0,C 180,E1 -666.581,E2 -666.581} C_VEL
LIN {X 0,Y 601.445,Z 346.564,A -85,B 0,C 180,E1 -669.535,E2 -669.535} C_VEL
LIN {X 0,Y 601.409,Z 346.568,A -85,B 0,C 180,E1 -672.59,E2 -672.59} C_VEL
LIN {X 0,Y 601.422,Z 346.566,A -85,B 0,C 180,E1 -674.534,E2 -674.534} C_VEL
LIN {X 0,Y 601.438,Z 346.565,A -85,B 0,C 180,E1 -677.405,E2 -677.405} C_VEL
LIN {X 0,Y 601.437,Z 346.564,A -85,B 0,C 180,E1 -680.463,E2 -680.463} C_VEL
LIN {X 0,Y 601.414,Z 346.567,A -85,B 0,C 180,E1 -683.417,E2 -683.417} C_VEL
LIN {X 0,Y 601.428,Z 346.563,A -85,B 0,C 180,E1 -686.063,E2 -686.063} C_VEL
LIN {X 0,Y 601.438,Z 346.566,A -85,B 0,C 180,E1 -688.54,E2 -688.54} C_VEL
LIN {X 0,Y 601.434,Z 346.564,A -85,B 0,C 180,E1 -691.373,E2 -691.373} C_VEL
LIN {X 0,Y 601.405,Z 346.566,A -85,B 0,C 180,E1 -693.636,E2 -693.636} C_VEL
LIN {X 0,Y 601.416,Z 346.571,A -85,B 0,C 180,E1 -696.589,E2 -696.589} C_VEL
LIN {X 0,Y 601.429,Z 346.563,A -85,B 0,C 180,E1 -699.478,E2 -699.478} C_VEL
LIN {X 0,Y 601.398,Z 346.57,A -85,B 0,C 180,E1 -702.311,E2 -702.311} C_VEL
LIN {X 0,Y 601.414,Z 346.57,A -85,B 0,C 180,E1 -704.408,E2 -704.408} C_VEL
LIN {X 0,Y 601.421,Z 346.566,A -85,B 0,C 180,E1 -707.172,E2 -707.172} C_VEL
LIN {X 0,Y 601.428,Z 346.563,A -85,B 0,C 180,E1 -709.905,E2 -709.905} C_VEL
LIN {X 0,Y 601.445,Z 346.571,A -85,B 0,C 180,E1 -712.615,E2 -712.615} C_VEL
LIN {X 0,Y 601.427,Z 346.563,A -85,B 0,C 180,E1 -715.308,E2 -715.308} C_VEL
LIN {X 0,Y 601.418,Z 346.566,A -85,B 0,C 180,E1 -717.991,E2 -717.991} C_VEL
LIN {X 0,Y 601.449,Z 346.568,A -85,B 0,C 180,E1 -720.669,E2 -720.669} C_VEL
LIN {X 0,Y 601.428,Z 346.563,A -85,B 0,C 180,E1 -723.349,E2 -723.349} C_VEL
LIN {X 0,Y 601.404,Z 346.569,A -85,B 0,C 180,E1 -726.037,E2 -726.037} C_VEL
LIN {X 0,Y 601.434,Z 346.567,A -85,B 0,C 180,E1 -728.738,E2 -728.738} C_VEL
LIN {X 0,Y 601.427,Z 346.562,A -85,B 0,C 180,E1 -731.458,E2 -731.458} C_VEL
LIN {X 0,Y 601.41,Z 346.572,A -85,B 0,C 180,E1 -734.206,E2 -734.206} C_VEL
LIN {X 0,Y 601.427,Z 346.564,A -85,B 0,C 180,E1 -736.986,E2 -736.986} C_VEL
LIN {X 0,Y 601.404,Z 346.568,A -85,B 0,C 180,E1 -739.809,E2 -739.809} C_VEL
LIN {X 0,Y 601.41,Z 346.568,A -85,B 0,C 180,E1 -742.683,E2 -742.683} C_VEL
LIN {X 0,Y 601.398,Z 346.567,A -85,B 0,C 180,E1 -744.879,E2 -744.879} C_VEL
LIN {X 0,Y 601.419,Z 346.568,A -85,B 0,C 180,E1 -747.867,E2 -747.867} C_VEL
LIN {X 0,Y 601.441,Z 346.571,A -85,B 0,C 180,E1 -750.163,E2 -750.163} C_VEL
LIN {X 0,Y 601.423,Z 346.565,A -85,B 0,C 180,E1 -752.718,E2 -752.718} C_VEL
LIN {X 0,Y 601.404,Z 346.565,A -85,B 0,C 180,E1 -755.115,E2 -755.115} C_VEL
LIN {X 0,Y 601.431,Z 346.563,A -85,B 0,C 180,E1 -757.419,E2 -757.419} C_VEL
LIN {X 0,Y 601.41,Z 346.574,A -85,B 0,C 180,E1 -759.995,E2 -759.995} C_VEL
LIN {X 0,Y 601.411,Z 346.566,A -85,B 0,C 180,E1 -762.67,E2 -762.67} C_VEL
LIN {X 0,Y 601.421,Z 346.566,A -85,B 0,C 180,E1 -765.483,E2 -765.483} C_VEL
LIN {X 0,Y 601.422,Z 346.567,A -85,B 0,C 180,E1 -768.407,E2 -768.407} C_VEL
LIN {X 0,Y 601.434,Z 346.562,A -85,B 0,C 180,E1 -770.876,E2 -770.876} C_VEL
LIN {X 0,Y 601.443,Z 346.568,A -85,B 0,C 180,E1 -773.734,E2 -773.734} C_VEL
LIN {X 0,Y 601.433,Z 346.569,A -85,B 0,C 180,E1 -776.065,E2 -776.065} C_VEL
LIN {X 0,Y 601.441,Z 346.562,A -85,B 0,C 180,E1 -778.542,E2 -778.542} C_VEL
LIN {X 0,Y 601.436,Z 346.565,A -85,B 0,C 180,E1 -781.374,E2 -781.374} C_VEL
LIN {X 0,Y 601.414,Z 346.57,A -85,B 0,C 180,E1 -784.133,E2 -784.133} C_VEL
LIN {X 0,Y 601.427,Z 346.655,A -85,B 0,C 180,E1 -786.75,E2 -786.75} C_VEL
LIN {X 0,Y 601.715,Z 351.666,A -85,B 0,C 180,E1 -787.446,E2 -787.446} C_VEL
LIN {X 0,Y 601.599,Z 372.083,A -85,B 0,C 180,E1 -790.198,E2 -790.198} C_VEL
LIN {X 0,Y 601.547,Z 393.356,A -85,B 0,C 180,E1 -793.018,E2 -793.018} C_VEL
LIN {X 0,Y 601.504,Z 416.28,A -85,B 0,C 180,E1 -796.011,E2 -796.011} C_VEL
LIN {X 0,Y 601.469,Z 422.524,A -85,B 0,C 180,E1 -796.819,E2 -796.819} C_VEL
LIN {X 0,Y 601.662,Z 439.266,A -85,B 0,C 180,E1 -797.027,E2 -797.027} C_VEL
LIN {X 0,Y 601.605,Z 530.962,A -85,B 0,C 180,E1 -798.14,E2 -798.14} C_VEL
LIN {X 0,Y 601.574,Z 544.227,A -85,B 0,C 180,E1 -798.438,E2 -798.438} C_VEL
LIN {X 0,Y 601.54,Z 556.706,A -85,B 0,C 180,E1 -798.856,E2 -798.856} C_VEL
LIN {X 0,Y 601.523,Z 568.638,A -85,B 0,C 180,E1 -799.396,E2 -799.396} C_VEL
LIN {X 0,Y 601.481,Z 580.202,A -85,B 0,C 180,E1 -800.076,E2 -800.076} C_VEL
LIN {X 0,Y 601.444,Z 590.598,A -85,B 0,C 180,E1 -800.839,E2 -800.839} C_VEL
LIN {X 0,Y 601.429,Z 599.114,A -85,B 0,C 180,E1 -801.601,E2 -801.601} C_VEL
LIN {X 0,Y 601.418,Z 606.962,A -85,B 0,C 180,E1 -802.446,E2 -802.446} C_VEL
LIN {X 0,Y 601.37,Z 614.225,A -85,B 0,C 180,E1 -803.398,E2 -803.398} C_VEL
LIN {X 0,Y 601.372,Z 619.867,A -85,B 0,C 180,E1 -804.299,E2 -804.299} C_VEL
LIN {X 0,Y 601.337,Z 624.95,A -85,B 0,C 180,E1 -805.307,E2 -805.307} C_VEL
LIN {X 0,Y 601.367,Z 628.896,A -85,B 0,C 180,E1 -806.315,E2 -806.315} C_VEL
LIN {X 0,Y 601.325,Z 631.809,A -85,B 0,C 180,E1 -807.321,E2 -807.321} C_VEL
LIN {X 0,Y 601.341,Z 633.202,A -85,B 0,C 180,E1 -807.991,E2 -807.991} C_VEL
LIN {X 0,Y 601.339,Z 634.784,A -85,B 0,C 180,E1 -809.33,E2 -809.33} C_VEL
LIN {X 0,Y 601.335,Z 635,A -85,B 0,C 180,E1 -810,E2 -810} C_VEL
LIN {X 0,Y 601.348,Z 634.184,A -85,B 0,C 180,E1 -811.339,E2 -811.339} C_VEL
LIN {X 0,Y 601.341,Z 633.202,A -85,B 0,C 180,E1 -812.009,E2 -812.009} C_VEL
LIN {X 0,Y 601.325,Z 631.809,A -85,B 0,C 180,E1 -812.679,E2 -812.679} C_VEL
LIN {X 0,Y 601.367,Z 628.896,A -85,B 0,C 180,E1 -813.685,E2 -813.685} C_VEL
LIN {X 0,Y 601.337,Z 624.95,A -85,B 0,C 180,E1 -814.693,E2 -814.693} C_VEL
LIN {X 0,Y 601.372,Z 618.878,A -85,B 0,C 180,E1 -815.869,E2 -815.869} C_VEL
LIN {X 0,Y 601.381,Z 612.237,A -85,B 0,C 180,E1 -816.88,E2 -816.88} C_VEL
LIN {X 0,Y 601.4,Z 603.991,A -85,B 0,C 180,E1 -817.892,E2 -817.892} C_VEL
LIN {X 0,Y 601.436,Z 595.539,A -85,B 0,C 180,E1 -818.737,E2 -818.737} C_VEL
LIN {X 0,Y 601.442,Z 585.095,A -85,B 0,C 180,E1 -819.585,E2 -819.585} C_VEL
LIN {X 0,Y 601.472,Z 574.761,A -85,B 0,C 180,E1 -820.264,E2 -820.264} C_VEL
LIN {X 0,Y 601.536,Z 563.907,A -85,B 0,C 180,E1 -820.835,E2 -820.835} C_VEL
LIN {X 0,Y 601.556,Z 551.385,A -85,B 0,C 180,E1 -821.34,E2 -821.34} C_VEL
LIN {X 0,Y 601.568,Z 538.363,A -85,B 0,C 180,E1 -821.711,E2 -821.711} C_VEL
LIN {X 0,Y 601.614,Z 525.105,A -85,B 0,C 180,E1 -821.946,E2 -821.946} C_VEL
LIN {X 0,Y 601.548,Z 423.168,A -85,B 0,C 180,E1 -823.169,E2 -823.169} C_VEL
LIN {X 0,Y 601.467,Z 422.275,A -85,B 0,C 180,E1 -823.213,E2 -823.213} C_VEL
LIN {X 0,Y 601.52,Z 400.004,A -85,B 0,C 180,E1 -826.11,E2 -826.11} C_VEL
LIN {X 0,Y 601.606,Z 377.402,A -85,B 0,C 180,E1 -829.092,E2 -829.092} C_VEL
LIN {X 0,Y 601.677,Z 356.128,A -85,B 0,C 180,E1 -831.948,E2 -831.948} C_VEL
LIN {X 0,Y 601.691,Z 348.151,A -85,B 0,C 180,E1 -833.034,E2 -833.034} C_VEL
LIN {X 0,Y 601.414,Z 346.569,A -85,B 0,C 180,E1 -833.273,E2 -833.273} C_VEL
LIN {X 0,Y 601.414,Z 346.57,A -85,B 0,C 180,E1 -835.867,E2 -835.867} C_VEL
LIN {X 0,Y 601.435,Z 346.565,A -85,B 0,C 180,E1 -838.626,E2 -838.626} C_VEL
LIN {X 0,Y 601.441,Z 346.562,A -85,B 0,C 180,E1 -841.458,E2 -841.458} C_VEL
LIN {X 0,Y 601.432,Z 346.572,A -85,B 0,C 180,E1 -844.117,E2 -844.117} C_VEL
LIN {X 0,Y 601.412,Z 346.567,A -85,B 0,C 180,E1 -846.581,E2 -846.581} C_VEL
LIN {X 0,Y 601.44,Z 346.564,A -85,B 0,C 180,E1 -849.535,E2 -849.535} C_VEL
LIN {X 0,Y 601.425,Z 346.57,A -85,B 0,C 180,E1 -851.764,E2 -851.764} C_VEL
LIN {X 0,Y 601.419,Z 346.565,A -85,B 0,C 180,E1 -854.534,E2 -854.534} C_VEL
LIN {X 0,Y 601.411,Z 346.567,A -85,B 0,C 180,E1 -857.33,E2 -857.33} C_VEL
LIN {X 0,Y 601.411,Z 346.573,A -85,B 0,C 180,E1 -860.005,E2 -860.005} C_VEL
LIN {X 0,Y 601.432,Z 346.562,A -85,B 0,C 180,E1 -862.617,E2 -862.617} C_VEL
LIN {X 0,Y 601.426,Z 346.563,A -85,B 0,C 180,E1 -865.069,E2 -865.069} C_VEL
LIN {X 0,Y 601.429,Z 346.568,A -85,B 0,C 180,E1 -867.484,E2 -867.484} C_VEL
LIN {X 0,Y 601.441,Z 346.569,A -85,B 0,C 180,E1 -869.847,E2 -869.847} C_VEL
LIN {X 0,Y 601.413,Z 346.564,A -85,B 0,C 180,E1 -872.636,E2 -872.636} C_VEL
LIN {X 0,Y 601.397,Z 346.568,A -85,B 0,C 180,E1 -875.121,E2 -875.121} C_VEL
LIN {X 0,Y 601.408,Z 346.571,A -85,B 0,C 180,E1 -877.393,E2 -877.393} C_VEL
LIN {X 0,Y 601.403,Z 346.567,A -85,B 0,C 180,E1 -880.191,E2 -880.191} C_VEL
LIN {X 0,Y 601.428,Z 346.564,A -85,B 0,C 180,E1 -883.014,E2 -883.014} C_VEL
LIN {X 0,Y 601.412,Z 346.568,A -85,B 0,C 180,E1 -885.907,E2 -885.907} C_VEL
LIN {X 0,Y 601.427,Z 346.562,A -85,B 0,C 180,E1 -888.542,E2 -888.542} C_VEL
LIN {X 0,Y 601.437,Z 346.569,A -85,B 0,C 180,E1 -891.263,E2 -891.263} C_VEL
LIN {X 0,Y 601.405,Z 346.567,A -85,B 0,C 180,E1 -893.963,E2 -893.963} C_VEL
LIN {X 0,Y 601.429,Z 346.563,A -85,B 0,C 180,E1 -896.651,E2 -896.651} C_VEL
LIN {X 0,Y 601.455,Z 346.57,A -85,B 0,C 180,E1 -899.331,E2 -899.331} C_VEL
LIN {X 0,Y 601.418,Z 346.564,A -85,B 0,C 180,E1 -902.009,E2 -902.009} C_VEL
LIN {X 0,Y 601.43,Z 346.564,A -85,B 0,C 180,E1 -904.692,E2 -904.692} C_VEL
LIN {X 0,Y 601.449,Z 346.568,A -85,B 0,C 180,E1 -907.385,E2 -907.385} C_VEL
LIN {X 0,Y 601.429,Z 346.562,A -85,B 0,C 180,E1 -910.095,E2 -910.095} C_VEL
LIN {X 0,Y 601.406,Z 346.565,A -85,B 0,C 180,E1 -912.39,E2 -912.39} C_VEL
LIN {X 0,Y 600.748,Z 346.655,A -85,B 0,C 180,E1 -912.949,E2 -912.949} C_VEL
LIN {X 0,Y 597.9,Z 347.013,A -85,B 0,C 180,E1 -913.857,E2 -913.857} C_VEL
LIN {X 0,Y 595.487,Z 347.314,A -85,B 0,C 180,E1 -914.587,E2 -914.587} C_VEL
LIN {X 0,Y 594.448,Z 347.442,A -85,B 0,C 180,E1 -915.151,E2 -915.151} C_VEL
LIN {X 0,Y 594.362,Z 347.448,A -85,B 0,C 180,E1 -915.341,E2 -915.341} C_VEL
LIN {X 0,Y 594.378,Z 347.441,A -85,B 0,C 180,E1 -917.905,E2 -917.905} C_VEL
LIN {X 0,Y 594.38,Z 347.448,A -85,B 0,C 180,E1 -920.92,E2 -920.92} C_VEL
LIN {X 0,Y 594.386,Z 347.44,A -85,B 0,C 180,E1 -923.705,E2 -923.705} C_VEL
LIN {X 0,Y 594.389,Z 347.445,A -85,B 0,C 180,E1 -926.7,E2 -926.7} C_VEL
LIN {X 0,Y 594.382,Z 347.45,A -85,B 0,C 180,E1 -928.999,E2 -928.999} C_VEL
LIN {X 0,Y 594.39,Z 347.44,A -85,B 0,C 180,E1 -931.647,E2 -931.647} C_VEL
LIN {X 0,Y 594.395,Z 347.443,A -85,B 0,C 180,E1 -934.579,E2 -934.579} C_VEL
LIN {X 0,Y 594.384,Z 347.446,A -85,B 0,C 180,E1 -937.087,E2 -937.087} C_VEL
LIN {X 0,Y 594.373,Z 347.441,A -85,B 0,C 180,E1 -939.776,E2 -939.776} C_VEL
LIN {X 0,Y 594.386,Z 347.443,A -85,B 0,C 180,E1 -942.374,E2 -942.374} C_VEL
LIN {X 0,Y 594.361,Z 347.446,A -85,B 0,C 180,E1 -945.192,E2 -945.192} C_VEL
LIN {X 0,Y 594.366,Z 347.442,A -85,B 0,C 180,E1 -947.626,E2 -947.626} C_VEL
LIN {X 0,Y 594.394,Z 347.444,A -85,B 0,C 180,E1 -950.322,E2 -950.322} C_VEL
LIN {X 0,Y 594.388,Z 347.446,A -85,B 0,C 180,E1 -952.914,E2 -952.914} C_VEL
LIN {X 0,Y 594.406,Z 347.57,A -85,B 0,C 180,E1 -955.859,E2 -955.859} C_VEL
LIN {X 0,Y 594.409,Z 361.353,A -85,B 0,C 180,E1 -958.353,E2 -958.353} C_VEL
LIN {X 0,Y 594.364,Z 374.764,A -85,B 0,C 180,E1 -960.734,E2 -960.734} C_VEL
LIN {X 0,Y 594.773,Z 379.105,A -85,B 0,C 180,E1 -960.796,E2 -960.796} C_VEL
LIN {X 0,Y 594.667,Z 480.9,A -85,B 0,C 180,E1 -962.043,E2 -962.043} C_VEL
LIN {X 0,Y 594.602,Z 494.443,A -85,B 0,C 180,E1 -962.352,E2 -962.352} C_VEL
LIN {X 0,Y 594.554,Z 507.199,A -85,B 0,C 180,E1 -962.787,E2 -962.787} C_VEL
LIN {X 0,Y 594.511,Z 518.497,A -85,B 0,C 180,E1 -963.307,E2 -963.307} C_VEL
LIN {X 0,Y 594.479,Z 529.568,A -85,B 0,C 180,E1 -963.96,E2 -963.96} C_VEL
LIN {X 0,Y 594.423,Z 541.028,A -85,B 0,C 180,E1 -964.81,E2 -964.81} C_VEL
LIN {X 0,Y 594.349,Z 551.072,A -85,B 0,C 180,E1 -965.746,E2 -965.746} C_VEL
LIN {X 0,Y 594.313,Z 559.064,A -85,B 0,C 180,E1 -966.663,E2 -966.663} C_VEL
LIN {X 0,Y 594.311,Z 566.849,A -85,B 0,C 180,E1 -967.765,E2 -967.765} C_VEL
LIN {X 0,Y 594.26,Z 572.801,A -85,B 0,C 180,E1 -968.837,E2 -968.837} C_VEL
LIN {X 0,Y 594.24,Z 577.554,A -85,B 0,C 180,E1 -969.942,E2 -969.942} C_VEL
LIN {X 0,Y 594.246,Z 581.232,A -85,B 0,C 180,E1 -971.111,E2 -971.111} C_VEL
LIN {X 0,Y 594.209,Z 583.331,A -85,B 0,C 180,E1 -972.091,E2 -972.091} C_VEL
LIN {X 0,Y 594.238,Z 584.761,A -85,B 0,C 180,E1 -973.333,E2 -973.333} C_VEL
LIN {X 0,Y 594.225,Z 584.967,A -85,B 0,C 180,E1 -974.216,E2 -974.216} C_VEL
LIN {X 0,Y 594.211,Z 584.65,A -85,B 0,C 180,E1 -974.918,E2 -974.918} C_VEL
LIN {X 0,Y 594.264,Z 583.529,A -85,B 0,C 180,E1 -975.877,E2 -975.877} C_VEL
LIN {X 0,Y 594.246,Z 581.138,A -85,B 0,C 180,E1 -977.015,E2 -977.015} C_VEL
LIN {X 0,Y 594.265,Z 577.888,A -85,B 0,C 180,E1 -978.056,E2 -978.056} C_VEL
LIN {X 0,Y 594.246,Z 573.561,A -85,B 0,C 180,E1 -979.093,E2 -979.093} C_VEL
LIN {X 0,Y 594.309,Z 567.01,A -85,B 0,C 180,E1 -980.299,E2 -980.299} C_VEL
LIN {X 0,Y 594.323,Z 559.847,A -85,B 0,C 180,E1 -981.329,E2 -981.329} C_VEL
LIN {X 0,Y 594.348,Z 550.96,A -85,B 0,C 180,E1 -982.356,E2 -982.356} C_VEL
LIN {X 0,Y 594.424,Z 541.873,A -85,B 0,C 180,E1 -983.21,E2 -983.21} C_VEL
LIN {X 0,Y 594.471,Z 531.835,A -85,B 0,C 180,E1 -983.977,E2 -983.977} C_VEL
LIN {X 0,Y 594.488,Z 520.781,A -85,B 0,C 180,E1 -984.658,E2 -984.658} C_VEL
LIN {X 0,Y 594.56,Z 508.403,A -85,B 0,C 180,E1 -985.254,E2 -985.254} C_VEL
LIN {X 0,Y 594.585,Z 495.804,A -85,B 0,C 180,E1 -985.7,E2 -985.7} C_VEL
LIN {X 0,Y 594.645,Z 482.421,A -85,B 0,C 180,E1 -986.019,E2 -986.019} C_VEL
LIN {X 0,Y 594.682,Z 449.438,A -85,B 0,C 180,E1 -986.443,E2 -986.443} C_VEL
LIN {X 0,Y 594.616,Z 376.233,A -85,B 0,C 180,E1 -987.333,E2 -987.333} C_VEL
LIN {X 0,Y 594.359,Z 374.569,A -85,B 0,C 180,E1 -987.374,E2 -987.374} C_VEL
LIN {X 0,Y 594.42,Z 359.887,A -85,B 0,C 180,E1 -990,E2 -990} C_VEL
LIN {X 0,Y 594.394,Z 347.442,A -85,B 0,C 180,E1 -992.266,E2 -992.266} C_VEL
LIN {X 0,Y 594.39,Z 347.441,A -85,B 0,C 180,E1 -994.748,E2 -994.748} C_VEL
LIN {X 0,Y 594.401,Z 347.448,A -85,B 0,C 180,E1 -997.473,E2 -997.473} C_VEL
LIN {X 0,Y 594.397,Z 347.439,A -85,B 0,C 180,E1 -1000.216,E2 -1000.216} C_VEL
LIN {X 0,Y 594.37,Z 347.446,A -85,B 0,C 180,E1 -1002.983,E2 -1002.983} C_VEL
LIN {X 0,Y 594.377,Z 347.446,A -85,B 0,C 180,E1 -1005.077,E2 -1005.077} C_VEL
LIN {X 0,Y 594.386,Z 347.448,A -85,B 0,C 180,E1 -1007.193,E2 -1007.193} C_VEL
LIN {X 0,Y 594.377,Z 347.441,A -85,B 0,C 180,E1 -1010.053,E2 -1010.053} C_VEL
LIN {X 0,Y 594.369,Z 347.447,A -85,B 0,C 180,E1 -1012.966,E2 -1012.966} C_VEL
LIN {X 0,Y 594.381,Z 347.45,A -85,B 0,C 180,E1 -1015.192,E2 -1015.192} C_VEL
LIN {X 0,Y 594.389,Z 347.445,A -85,B 0,C 180,E1 -1017.526,E2 -1017.526} C_VEL
LIN {X 0,Y 594.39,Z 347.439,A -85,B 0,C 180,E1 -1020.328,E2 -1020.328} C_VEL
LIN {X 0,Y 594.379,Z 347.447,A -85,B 0,C 180,E1 -1022.949,E2 -1022.949} C_VEL
LIN {X 0,Y 594.386,Z 347.445,A -85,B 0,C 180,E1 -1025.406,E2 -1025.406} C_VEL
LIN {X 0,Y 594.387,Z 347.44,A -85,B 0,C 180,E1 -1027.94,E2 -1027.94} C_VEL
LIN {X 0,Y 594.378,Z 347.447,A -85,B 0,C 180,E1 -1030.821,E2 -1030.821} C_VEL
LIN {X 0,Y 594.38,Z 347.441,A -85,B 0,C 180,E1 -1033.84,E2 -1033.84} C_VEL
LIN {X 0,Y 594.384,Z 347.445,A -85,B 0,C 180,E1 -1036.702,E2 -1036.702} C_VEL
LIN {X 0,Y 594.373,Z 347.444,A -85,B 0,C 180,E1 -1039.433,E2 -1039.433} C_VEL
LIN {X 0,Y 594.388,Z 347.441,A -85,B 0,C 180,E1 -1042.39,E2 -1042.39} C_VEL
LIN {X 0,Y 594.378,Z 347.447,A -85,B 0,C 180,E1 -1044.671,E2 -1044.671} C_VEL
LIN {X 0,Y 594.376,Z 347.448,A -85,B 0,C 180,E1 -1047.087,E2 -1047.087} C_VEL
LIN {X 0,Y 594.381,Z 347.441,A -85,B 0,C 180,E1 -1049.67,E2 -1049.67} C_VEL
LIN {X 0,Y 594.384,Z 347.445,A -85,B 0,C 180,E1 -1052.539,E2 -1052.539} C_VEL
LIN {X 0,Y 594.373,Z 347.452,A -85,B 0,C 180,E1 -1054.806,E2 -1054.806} C_VEL
LIN {X 0,Y 594.364,Z 347.445,A -85,B 0,C 180,E1 -1057.262,E2 -1057.262} C_VEL
LIN {X 0,Y 594.374,Z 347.441,A -85,B 0,C 180,E1 -1059.946,E2 -1059.946} C_VEL
LIN {X 0,Y 594.387,Z 347.449,A -85,B 0,C 180,E1 -1062.806,E2 -1062.806} C_VEL
LIN {X 0,Y 594.38,Z 347.441,A -85,B 0,C 180,E1 -1065.825,E2 -1065.825} C_VEL
LIN {X 0,Y 594.386,Z 347.446,A -85,B 0,C 180,E1 -1068.404,E2 -1068.404} C_VEL
LIN {X 0,Y 594.396,Z 347.441,A -85,B 0,C 180,E1 -1071.158,E2 -1071.158} C_VEL
LIN {X 0,Y 594.36,Z 347.444,A -85,B 0,C 180,E1 -1073.891,E2 -1073.891} C_VEL
LIN {X 0,Y 594.38,Z 347.45,A -85,B 0,C 180,E1 -1076.61,E2 -1076.61} C_VEL
LIN {X 0,Y 594.417,Z 347.436,A -85,B 0,C 180,E1 -1079.322,E2 -1079.322} C_VEL
LIN {X 0,Y 594.388,Z 347.442,A -85,B 0,C 180,E1 -1082.033,E2 -1082.033} C_VEL
LIN {X 0,Y 594.394,Z 347.444,A -85,B 0,C 180,E1 -1084.747,E2 -1084.747} C_VEL
LIN {X 0,Y 594.394,Z 347.439,A -85,B 0,C 180,E1 -1087.473,E2 -1087.473} C_VEL
LIN {X 0,Y 594.388,Z 347.446,A -85,B 0,C 180,E1 -1090.216,E2 -1090.216} C_VEL
LIN {X 0,Y 594.365,Z 347.444,A -85,B 0,C 180,E1 -1092.983,E2 -1092.983} C_VEL
LIN {X 0,Y 594.366,Z 347.444,A -85,B 0,C 180,E1 -1095.781,E2 -1095.781} C_VEL
LIN {X 0,Y 594.38,Z 347.446,A -85,B 0,C 180,E1 -1098.618,E2 -1098.618} C_VEL
LIN {X 0,Y 594.365,Z 347.443,A -85,B 0,C 180,E1 -1101.503,E2 -1101.503} C_VEL
LIN {X 0,Y 594.38,Z 347.447,A -85,B 0,C 180,E1 -1104.446,E2 -1104.446} C_VEL
LIN {X 0,Y 594.382,Z 347.443,A -85,B 0,C 180,E1 -1106.7,E2 -1106.7} C_VEL
LIN {X 0,Y 594.377,Z 347.441,A -85,B 0,C 180,E1 -1108.999,E2 -1108.999} C_VEL
LIN {X 0,Y 594.388,Z 347.442,A -85,B 0,C 180,E1 -1111.646,E2 -1111.646} C_VEL
LIN {X 0,Y 594.388,Z 347.443,A -85,B 0,C 180,E1 -1114.58,E2 -1114.58} C_VEL
LIN {X 0,Y 594.381,Z 347.44,A -85,B 0,C 180,E1 -1117.087,E2 -1117.087} C_VEL
LIN {X 0,Y 594.373,Z 347.446,A -85,B 0,C 180,E1 -1119.776,E2 -1119.776} C_VEL
LIN {X 0,Y 594.369,Z 347.447,A -85,B 0,C 180,E1 -1122.375,E2 -1122.375} C_VEL
LIN {X 0,Y 594.358,Z 347.443,A -85,B 0,C 180,E1 -1125.192,E2 -1125.192} C_VEL
LIN {X 0,Y 594.367,Z 347.446,A -85,B 0,C 180,E1 -1127.626,E2 -1127.626} C_VEL
LIN {X 0,Y 594.393,Z 347.443,A -85,B 0,C 180,E1 -1130.322,E2 -1130.322} C_VEL
LIN {X 0,Y 594.384,Z 347.44,A -85,B 0,C 180,E1 -1132.914,E2 -1132.914} C_VEL
LIN {X 0,Y 594.386,Z 347.45,A -85,B 0,C 180,E1 -1135.861,E2 -1135.861} C_VEL
LIN {X 0,Y 594.391,Z 347.44,A -85,B 0,C 180,E1 -1138.652,E2 -1138.652} C_VEL
LIN {X 0,Y 594.384,Z 347.441,A -85,B 0,C 180,E1 -1141.042,E2 -1141.042} C_VEL
LIN {X 0,Y 594.389,Z 347.448,A -85,B 0,C 180,E1 -1143.977,E2 -1143.977} C_VEL
LIN {X 0,Y 594.393,Z 347.486,A -85,B 0,C 180,E1 -1146.574,E2 -1146.574} C_VEL
LIN {X 0,Y 594.802,Z 351.635,A -85,B 0,C 180,E1 -1147.165,E2 -1147.165} C_VEL
LIN {X 0,Y 594.67,Z 372.083,A -85,B 0,C 180,E1 -1149.957,E2 -1149.957} C_VEL
LIN {X 0,Y 594.572,Z 392.027,A -85,B 0,C 180,E1 -1152.635,E2 -1152.635} C_VEL
LIN {X 0,Y 594.484,Z 414.63,A -85,B 0,C 180,E1 -1155.626,E2 -1155.626} C_VEL
LIN {X 0,Y 594.46,Z 422.524,A -85,B 0,C 180,E1 -1156.661,E2 -1156.661} C_VEL
LIN {X 0,Y 594.783,Z 428.534,A -85,B 0,C 180,E1 -1156.744,E2 -1156.744} C_VEL
LIN {X 0,Y 594.684,Z 530.961,A -85,B 0,C 180,E1 -1158,E2 -1158} C_VEL
LIN {X 0,Y 594.616,Z 544.227,A -85,B 0,C 180,E1 -1158.301,E2 -1158.301} C_VEL
LIN {X 0,Y 594.569,Z 557.413,A -85,B 0,C 180,E1 -1158.75,E2 -1158.75} C_VEL
LIN {X 0,Y 594.537,Z 568.637,A -85,B 0,C 180,E1 -1159.27,E2 -1159.27} C_VEL
LIN {X 0,Y 594.469,Z 580.203,A -85,B 0,C 180,E1 -1159.958,E2 -1159.958} C_VEL
LIN {X 0,Y 594.413,Z 590.599,A -85,B 0,C 180,E1 -1160.73,E2 -1160.73} C_VEL
LIN {X 0,Y 594.383,Z 599.114,A -85,B 0,C 180,E1 -1161.501,E2 -1161.501} C_VEL
LIN {X 0,Y 594.347,Z 606.962,A -85,B 0,C 180,E1 -1162.356,E2 -1162.356} C_VEL
LIN {X 0,Y 594.282,Z 614.813,A -85,B 0,C 180,E1 -1163.408,E2 -1163.408} C_VEL
LIN {X 0,Y 594.289,Z 621.681,A -85,B 0,C 180,E1 -1164.571,E2 -1164.571} C_VEL
LIN {X 0,Y 594.27,Z 626.372,A -85,B 0,C 180,E1 -1165.591,E2 -1165.591} C_VEL
LIN {X 0,Y 594.267,Z 629.957,A -85,B 0,C 180,E1 -1166.61,E2 -1166.61} C_VEL
LIN {X 0,Y 594.226,Z 631.809,A -85,B 0,C 180,E1 -1167.288,E2 -1167.288} C_VEL
LIN {X 0,Y 594.24,Z 633.201,A -85,B 0,C 180,E1 -1167.967,E2 -1167.967} C_VEL
LIN {X 0,Y 594.239,Z 634.784,A -85,B 0,C 180,E1 -1169.322,E2 -1169.322} C_VEL
LIN {X 0,Y 594.236,Z 635,A -85,B 0,C 180,E1 -1170,E2 -1170} C_VEL
LIN {X 0,Y 594.247,Z 634.185,A -85,B 0,C 180,E1 -1171.355,E2 -1171.355} C_VEL
LIN {X 0,Y 594.24,Z 633.202,A -85,B 0,C 180,E1 -1172.033,E2 -1172.033} C_VEL
LIN {X 0,Y 594.226,Z 631.81,A -85,B 0,C 180,E1 -1172.712,E2 -1172.712} C_VEL
LIN {X 0,Y 594.288,Z 628.896,A -85,B 0,C 180,E1 -1173.729,E2 -1173.729} C_VEL
LIN {X 0,Y 594.242,Z 624.95,A -85,B 0,C 180,E1 -1174.749,E2 -1174.749} C_VEL
LIN {X 0,Y 594.304,Z 618.878,A -85,B 0,C 180,E1 -1175.939,E2 -1175.939} C_VEL
LIN {X 0,Y 594.308,Z 612.237,A -85,B 0,C 180,E1 -1176.962,E2 -1176.962} C_VEL
LIN {X 0,Y 594.359,Z 603.991,A -85,B 0,C 180,E1 -1177.986,E2 -1177.986} C_VEL
LIN {X 0,Y 594.382,Z 595.539,A -85,B 0,C 180,E1 -1178.842,E2 -1178.842} C_VEL
LIN {X 0,Y 594.427,Z 585.097,A -85,B 0,C 180,E1 -1179.699,E2 -1179.699} C_VEL
LIN {X 0,Y 594.482,Z 574.763,A -85,B 0,C 180,E1 -1180.386,E2 -1180.386} C_VEL
LIN {X 0,Y 594.559,Z 563.705,A -85,B 0,C 180,E1 -1180.974,E2 -1180.974} C_VEL
LIN {X 0,Y 594.582,Z 551.712,A -85,B 0,C 180,E1 -1181.464,E2 -1181.464} C_VEL
LIN {X 0,Y 594.637,Z 538.363,A -85,B 0,C 180,E1 -1181.85,E2 -1181.85} C_VEL
LIN {X 0,Y 594.693,Z 525.105,A -85,B 0,C 180,E1 -1182.087,E2 -1182.087} C_VEL
LIN {X 0,Y 594.652,Z 423.95,A -85,B 0,C 180,E1 -1183.315,E2 -1183.315} C_VEL
LIN {X 0,Y 594.448,Z 422.441,A -85,B 0,C 180,E1 -1183.35,E2 -1183.35} C_VEL
LIN {X 0,Y 594.533,Z 400.004,A -85,B 0,C 180,E1 -1186.305,E2 -1186.305} C_VEL
LIN {X 0,Y 594.67,Z 377.402,A -85,B 0,C 180,E1 -1189.324,E2 -1189.324} C_VEL
LIN {X 0,Y 594.807,Z 355.013,A -85,B 0,C 180,E1 -1192.369,E2 -1192.369} C_VEL
LIN {X 0,Y 594.758,Z 349.48,A -85,B 0,C 180,E1 -1193.135,E2 -1193.135} C_VEL
LIN {X 0,Y 594.38,Z 347.447,A -85,B 0,C 180,E1 -1193.45,E2 -1193.45} C_VEL
LIN {X 0,Y 594.389,Z 347.448,A -85,B 0,C 180,E1 -1196.023,E2 -1196.023} C_VEL
LIN {X 0,Y 594.384,Z 347.441,A -85,B 0,C 180,E1 -1198.958,E2 -1198.958} C_VEL
LIN {X 0,Y 594.392,Z 347.442,A -85,B 0,C 180,E1 -1201.645,E2 -1201.645} C_VEL
LIN {X 0,Y 594.399,Z 347.441,A -85,B 0,C 180,E1 -1204.578,E2 -1204.578} C_VEL
LIN {X 0,Y 594.384,Z 347.44,A -85,B 0,C 180,E1 -1207.086,E2 -1207.086} C_VEL
LIN {X 0,Y 594.376,Z 347.447,A -85,B 0,C 180,E1 -1209.774,E2 -1209.774} C_VEL
LIN {X 0,Y 594.366,Z 347.446,A -85,B 0,C 180,E1 -1212.374,E2 -1212.374} C_VEL
LIN {X 0,Y 594.358,Z 347.444,A -85,B 0,C 180,E1 -1215.191,E2 -1215.191} C_VEL
LIN {X 0,Y 594.369,Z 347.448,A -85,B 0,C 180,E1 -1217.625,E2 -1217.625} C_VEL
LIN {X 0,Y 594.388,Z 347.442,A -85,B 0,C 180,E1 -1220.32,E2 -1220.32} C_VEL
LIN {X 0,Y 594.381,Z 347.44,A -85,B 0,C 180,E1 -1222.913,E2 -1222.913} C_VEL
LIN {X 0,Y 594.379,Z 347.45,A -85,B 0,C 180,E1 -1225.86,E2 -1225.86} C_VEL
LIN {X 0,Y 594.385,Z 347.44,A -85,B 0,C 180,E1 -1228.651,E2 -1228.651} C_VEL
LIN {X 0,Y 594.378,Z 347.442,A -85,B 0,C 180,E1 -1231.041,E2 -1231.041} C_VEL
LIN {X 0,Y 594.383,Z 347.445,A -85,B 0,C 180,E1 -1233.975,E2 -1233.975} C_VEL
LIN {X 0,Y 594.383,Z 347.441,A -85,B 0,C 180,E1 -1236.296,E2 -1236.296} C_VEL
LIN {X 0,Y 594.4,Z 347.442,A -85,B 0,C 180,E1 -1239.224,E2 -1239.224} C_VEL
LIN {X 0,Y 594.375,Z 347.443,A -85,B 0,C 180,E1 -1242.096,E2 -1242.096} C_VEL
LIN {X 0,Y 594.365,Z 347.443,A -85,B 0,C 180,E1 -1244.219,E2 -1244.219} C_VEL
LIN {X 0,Y 594.366,Z 347.445,A -85,B 0,C 180,E1 -1247.017,E2 -1247.017} C_VEL
LIN {X 0,Y 594.389,Z 347.444,A -85,B 0,C 180,E1 -1249.784,E2 -1249.784} C_VEL
LIN {X 0,Y 594.394,Z 347.438,A -85,B 0,C 180,E1 -1252.527,E2 -1252.527} C_VEL
LIN {X 0,Y 594.4,Z 347.446,A -85,B 0,C 180,E1 -1255.253,E2 -1255.253} C_VEL
LIN {X 0,Y 594.389,Z 347.441,A -85,B 0,C 180,E1 -1257.967,E2 -1257.967} C_VEL
LIN {X 0,Y 594.421,Z 347.437,A -85,B 0,C 180,E1 -1260.678,E2 -1260.678} C_VEL
LIN {X 0,Y 594.385,Z 347.449,A -85,B 0,C 180,E1 -1263.389,E2 -1263.389} C_VEL
LIN {X 0,Y 594.361,Z 347.443,A -85,B 0,C 180,E1 -1266.109,E2 -1266.109} C_VEL
LIN {X 0,Y 594.41,Z 347.436,A -85,B 0,C 180,E1 -1268.157,E2 -1268.157} C_VEL
LIN {X 0,Y 594.389,Z 347.448,A -85,B 0,C 180,E1 -1271.08,E2 -1271.08} C_VEL
LIN {X 0,Y 594.38,Z 347.443,A -85,B 0,C 180,E1 -1273.679,E2 -1273.679} C_VEL
LIN {X 0,Y 594.362,Z 347.448,A -85,B 0,C 180,E1 -1275.341,E2 -1275.341} C_VEL
LIN {X 0,Y 593.692,Z 347.528,A -85,B 0,C 180,E1 -1275.907,E2 -1275.907} C_VEL
LIN {X 0,Y 590.836,Z 347.887,A -85,B 0,C 180,E1 -1276.825,E2 -1276.825} C_VEL
LIN {X 0,Y 588.43,Z 348.185,A -85,B 0,C 180,E1 -1277.564,E2 -1277.564} C_VEL
LIN {X 0,Y 587.402,Z 348.31,A -85,B 0,C 180,E1 -1278.134,E2 -1278.134} C_VEL
LIN {X 0,Y 587.322,Z 348.32,A -85,B 0,C 180,E1 -1278.327,E2 -1278.327} C_VEL
LIN {X 0,Y 587.35,Z 348.326,A -85,B 0,C 180,E1 -1281.046,E2 -1281.046} C_VEL
LIN {X 0,Y 587.36,Z 348.321,A -85,B 0,C 180,E1 -1283.257,E2 -1283.257} C_VEL
LIN {X 0,Y 587.358,Z 348.316,A -85,B 0,C 180,E1 -1286.278,E2 -1286.278} C_VEL
LIN {X 0,Y 587.348,Z 348.323,A -85,B 0,C 180,E1 -1289.135,E2 -1289.135} C_VEL
LIN {X 0,Y 587.353,Z 348.316,A -85,B 0,C 180,E1 -1291.839,E2 -1291.839} C_VEL
LIN {X 0,Y 587.353,Z 348.317,A -85,B 0,C 180,E1 -1294.35,E2 -1294.35} C_VEL
LIN {X 0,Y 587.35,Z 348.325,A -85,B 0,C 180,E1 -1296.747,E2 -1296.747} C_VEL
LIN {X 0,Y 587.343,Z 348.319,A -85,B 0,C 180,E1 -1299.36,E2 -1299.36} C_VEL
LIN {X 0,Y 587.334,Z 348.319,A -85,B 0,C 180,E1 -1302.109,E2 -1302.109} C_VEL
LIN {X 0,Y 587.314,Z 348.325,A -85,B 0,C 180,E1 -1305.09,E2 -1305.09} C_VEL
LIN {X 0,Y 587.352,Z 348.317,A -85,B 0,C 180,E1 -1307.929,E2 -1307.929} C_VEL
LIN {X 0,Y 587.336,Z 348.323,A -85,B 0,C 180,E1 -1311.059,E2 -1311.059} C_VEL
LIN {X 0,Y 587.355,Z 348.319,A -85,B 0,C 180,E1 -1313.292,E2 -1313.292} C_VEL
LIN {X 0,Y 587.378,Z 348.375,A -85,B 0,C 180,E1 -1315.782,E2 -1315.782} C_VEL
LIN {X 0,Y 587.388,Z 361.758,A -85,B 0,C 180,E1 -1318.235,E2 -1318.235} C_VEL
LIN {X 0,Y 587.324,Z 374.604,A -85,B 0,C 180,E1 -1320.56,E2 -1320.56} C_VEL
LIN {X 0,Y 587.868,Z 378.93,A -85,B 0,C 180,E1 -1320.635,E2 -1320.635} C_VEL
LIN {X 0,Y 587.737,Z 481.565,A -85,B 0,C 180,E1 -1321.912,E2 -1321.912} C_VEL
LIN {X 0,Y 587.636,Z 495.327,A -85,B 0,C 180,E1 -1322.237,E2 -1322.237} C_VEL
LIN {X 0,Y 587.601,Z 507.876,A -85,B 0,C 180,E1 -1322.679,E2 -1322.679} C_VEL
LIN {X 0,Y 587.516,Z 519.84,A -85,B 0,C 180,E1 -1323.252,E2 -1323.252} C_VEL
LIN {X 0,Y 587.453,Z 530.749,A -85,B 0,C 180,E1 -1323.919,E2 -1323.919} C_VEL
LIN {X 0,Y 587.388,Z 540.762,A -85,B 0,C 180,E1 -1324.676,E2 -1324.676} C_VEL
LIN {X 0,Y 587.33,Z 549.632,A -85,B 0,C 180,E1 -1325.494,E2 -1325.494} C_VEL
LIN {X 0,Y 587.272,Z 558.902,A -85,B 0,C 180,E1 -1326.553,E2 -1326.553} C_VEL
LIN {X 0,Y 587.241,Z 566.718,A -85,B 0,C 180,E1 -1327.668,E2 -1327.668} C_VEL
LIN {X 0,Y 587.184,Z 571.886,A -85,B 0,C 180,E1 -1328.59,E2 -1328.59} C_VEL
LIN {X 0,Y 587.191,Z 576.813,A -85,B 0,C 180,E1 -1329.691,E2 -1329.691} C_VEL
LIN {X 0,Y 587.156,Z 581.076,A -85,B 0,C 180,E1 -1331.015,E2 -1331.015} C_VEL
LIN {X 0,Y 587.13,Z 583.001,A -85,B 0,C 180,E1 -1331.868,E2 -1331.868} C_VEL
LIN {X 0,Y 587.148,Z 584.713,A -85,B 0,C 180,E1 -1333.253,E2 -1333.253} C_VEL
LIN {X 0,Y 587.139,Z 584.999,A -85,B 0,C 180,E1 -1334.02,E2 -1334.02} C_VEL
LIN {X 0,Y 587.125,Z 584.784,A -85,B 0,C 180,E1 -1334.732,E2 -1334.732} C_VEL
LIN {X 0,Y 587.162,Z 583.655,A -85,B 0,C 180,E1 -1335.82,E2 -1335.82} C_VEL
LIN {X 0,Y 587.148,Z 581.643,A -85,B 0,C 180,E1 -1336.855,E2 -1336.855} C_VEL
LIN {X 0,Y 587.175,Z 578.589,A -85,B 0,C 180,E1 -1337.91,E2 -1337.91} C_VEL
LIN {X 0,Y 587.169,Z 574.471,A -85,B 0,C 180,E1 -1338.959,E2 -1338.959} C_VEL
LIN {X 0,Y 587.202,Z 568.151,A -85,B 0,C 180,E1 -1340.18,E2 -1340.18} C_VEL
LIN {X 0,Y 587.266,Z 561.287,A -85,B 0,C 180,E1 -1341.224,E2 -1341.224} C_VEL
LIN {X 0,Y 587.282,Z 552.774,A -85,B 0,C 180,E1 -1342.263,E2 -1342.263} C_VEL
LIN {X 0,Y 587.389,Z 542.558,A -85,B 0,C 180,E1 -1343.26,E2 -1343.26} C_VEL
LIN {X 0,Y 587.462,Z 532.124,A -85,B 0,C 180,E1 -1344.078,E2 -1344.078} C_VEL
LIN {X 0,Y 587.485,Z 521.138,A -85,B 0,C 180,E1 -1344.767,E2 -1344.767} C_VEL
LIN {X 0,Y 587.599,Z 508.834,A -85,B 0,C 180,E1 -1345.369,E2 -1345.369} C_VEL
LIN {X 0,Y 587.64,Z 497.171,A -85,B 0,C 180,E1 -1345.799,E2 -1345.799} C_VEL
LIN {X 0,Y 587.704,Z 484.527,A -85,B 0,C 180,E1 -1346.122,E2 -1346.122} C_VEL
LIN {X 0,Y 587.741,Z 468.51,A -85,B 0,C 180,E1 -1346.358,E2 -1346.358} C_VEL
LIN {X 0,Y 587.782,Z 377.614,A -85,B 0,C 180,E1 -1347.473,E2 -1347.473} C_VEL
LIN {X 0,Y 587.334,Z 374.574,A -85,B 0,C 180,E1 -1347.535,E2 -1347.535} C_VEL
LIN {X 0,Y 587.389,Z 360.963,A -85,B 0,C 180,E1 -1350,E2 -1350} C_VEL
LIN {X 0,Y 587.37,Z 348.342,A -85,B 0,C 180,E1 -1352.314,E2 -1352.314} C_VEL
LIN {X 0,Y 587.365,Z 348.325,A -85,B 0,C 180,E1 -1355.493,E2 -1355.493} C_VEL
LIN {X 0,Y 587.348,Z 348.317,A -85,B 0,C 180,E1 -1358.255,E2 -1358.255} C_VEL
LIN {X 0,Y 587.355,Z 348.321,A -85,B 0,C 180,E1 -1361.133,E2 -1361.133} C_VEL
LIN {X 0,Y 587.372,Z 348.314,A -85,B 0,C 180,E1 -1364.26,E2 -1364.26} C_VEL
LIN {X 0,Y 587.351,Z 348.325,A -85,B 0,C 180,E1 -1367.405,E2 -1367.405} C_VEL
LIN {X 0,Y 587.331,Z 348.318,A -85,B 0,C 180,E1 -1370.304,E2 -1370.304} C_VEL
LIN {X 0,Y 587.326,Z 348.33,A -85,B 0,C 180,E1 -1373.258,E2 -1373.258} C_VEL
LIN {X 0,Y 587.339,Z 348.323,A -85,B 0,C 180,E1 -1375.516,E2 -1375.516} C_VEL
LIN {X 0,Y 587.349,Z 348.318,A -85,B 0,C 180,E1 -1377.817,E2 -1377.817} C_VEL
LIN {X 0,Y 587.345,Z 348.318,A -85,B 0,C 180,E1 -1380.51,E2 -1380.51} C_VEL
LIN {X 0,Y 587.34,Z 348.327,A -85,B 0,C 180,E1 -1383.111,E2 -1383.111} C_VEL
LIN {X 0,Y 587.358,Z 348.316,A -85,B 0,C 180,E1 -1385.894,E2 -1385.894} C_VEL
LIN {X 0,Y 587.334,Z 348.32,A -85,B 0,C 180,E1 -1388.478,E2 -1388.478} C_VEL
LIN {X 0,Y 587.336,Z 348.327,A -85,B 0,C 180,E1 -1391.156,E2 -1391.156} C_VEL
LIN {X 0,Y 587.332,Z 348.318,A -85,B 0,C 180,E1 -1394.113,E2 -1394.113} C_VEL
LIN {X 0,Y 587.335,Z 348.329,A -85,B 0,C 180,E1 -1396.995,E2 -1396.995} C_VEL
LIN {X 0,Y 587.32,Z 348.32,A -85,B 0,C 180,E1 -1399.98,E2 -1399.98} C_VEL
LIN {X 0,Y 587.343,Z 348.319,A -85,B 0,C 180,E1 -1402.392,E2 -1402.392} C_VEL
LIN {X 0,Y 587.344,Z 348.327,A -85,B 0,C 180,E1 -1404.945,E2 -1404.945} C_VEL
LIN {X 0,Y 587.338,Z 348.32,A -85,B 0,C 180,E1 -1407.42,E2 -1407.42} C_VEL
LIN {X 0,Y 587.329,Z 348.319,A -85,B 0,C 180,E1 -1409.829,E2 -1409.829} C_VEL
LIN {X 0,Y 587.345,Z 348.319,A -85,B 0,C 180,E1 -1412.306,E2 -1412.306} C_VEL
LIN {X 0,Y 587.332,Z 348.323,A -85,B 0,C 180,E1 -1414.483,E2 -1414.483} C_VEL
LIN {X 0,Y 587.339,Z 348.318,A -85,B 0,C 180,E1 -1417.486,E2 -1417.486} C_VEL
LIN {X 0,Y 587.328,Z 348.319,A -85,B 0,C 180,E1 -1419.695,E2 -1419.695} C_VEL
LIN {X 0,Y 587.354,Z 348.324,A -85,B 0,C 180,E1 -1422.594,E2 -1422.594} C_VEL
LIN {X 0,Y 587.356,Z 348.315,A -85,B 0,C 180,E1 -1425.739,E2 -1425.739} C_VEL
LIN {X 0,Y 587.353,Z 348.323,A -85,B 0,C 180,E1 -1428.858,E2 -1428.858} C_VEL
LIN {X 0,Y 587.363,Z 348.315,A -85,B 0,C 180,E1 -1431.744,E2 -1431.744} C_VEL
LIN {X 0,Y 587.354,Z 348.325,A -85,B 0,C 180,E1 -1434.507,E2 -1434.507} C_VEL
LIN {X 0,Y 587.374,Z 348.314,A -85,B 0,C 180,E1 -1437.257,E2 -1437.257} C_VEL
LIN {X 0,Y 587.373,Z 348.316,A -85,B 0,C 180,E1 -1440,E2 -1440} C_VEL
LIN {X 0,Y 587.374,Z 348.319,A -85,B 0,C 180,E1 -1442.743,E2 -1442.743} C_VEL
LIN {X 0,Y 587.352,Z 348.316,A -85,B 0,C 180,E1 -1445.493,E2 -1445.493} C_VEL
LIN {X 0,Y 587.363,Z 348.322,A -85,B 0,C 180,E1 -1448.255,E2 -1448.255} C_VEL
LIN {X 0,Y 587.352,Z 348.317,A -85,B 0,C 180,E1 -1451.141,E2 -1451.141} C_VEL
LIN {X 0,Y 587.355,Z 348.324,A -85,B 0,C 180,E1 -1454.261,E2 -1454.261} C_VEL
LIN {X 0,Y 587.352,Z 348.316,A -85,B 0,C 180,E1 -1457.406,E2 -1457.406} C_VEL
LIN {X 0,Y 587.327,Z 348.33,A -85,B 0,C 180,E1 -1460.305,E2 -1460.305} C_VEL
LIN {X 0,Y 587.318,Z 348.32,A -85,B 0,C 180,E1 -1463.259,E2 -1463.259} C_VEL
LIN {X 0,Y 587.354,Z 348.325,A -85,B 0,C 180,E1 -1466.183,E2 -1466.183} C_VEL
LIN {X 0,Y 587.345,Z 348.317,A -85,B 0,C 180,E1 -1469.135,E2 -1469.135} C_VEL
LIN {X 0,Y 587.351,Z 348.321,A -85,B 0,C 180,E1 -1471.839,E2 -1471.839} C_VEL
LIN {X 0,Y 587.349,Z 348.323,A -85,B 0,C 180,E1 -1474.35,E2 -1474.35} C_VEL
LIN {X 0,Y 587.347,Z 348.318,A -85,B 0,C 180,E1 -1476.747,E2 -1476.747} C_VEL
LIN {X 0,Y 587.342,Z 348.318,A -85,B 0,C 180,E1 -1479.36,E2 -1479.36} C_VEL
LIN {X 0,Y 587.329,Z 348.328,A -85,B 0,C 180,E1 -1482.108,E2 -1482.108} C_VEL
LIN {X 0,Y 587.311,Z 348.321,A -85,B 0,C 180,E1 -1484.912,E2 -1484.912} C_VEL
LIN {X 0,Y 587.317,Z 348.32,A -85,B 0,C 180,E1 -1486.995,E2 -1486.995} C_VEL
LIN {X 0,Y 587.326,Z 348.326,A -85,B 0,C 180,E1 -1489.748,E2 -1489.748} C_VEL
LIN {X 0,Y 587.344,Z 348.32,A -85,B 0,C 180,E1 -1492.393,E2 -1492.393} C_VEL
LIN {X 0,Y 587.351,Z 348.316,A -85,B 0,C 180,E1 -1494.947,E2 -1494.947} C_VEL
LIN {X 0,Y 587.34,Z 348.32,A -85,B 0,C 180,E1 -1497.422,E2 -1497.422} C_VEL
LIN {X 0,Y 587.348,Z 348.327,A -85,B 0,C 180,E1 -1499.831,E2 -1499.831} C_VEL
LIN {X 0,Y 587.352,Z 348.32,A -85,B 0,C 180,E1 -1502.307,E2 -1502.307} C_VEL
LIN {X 0,Y 587.336,Z 348.321,A -85,B 0,C 180,E1 -1504.484,E2 -1504.484} C_VEL
LIN {X 0,Y 587.387,Z 348.483,A -85,B 0,C 180,E1 -1506.418,E2 -1506.418} C_VEL
LIN {X 0,Y 587.915,Z 352.438,A -85,B 0,C 180,E1 -1506.995,E2 -1506.995} C_VEL
LIN {X 0,Y 587.737,Z 373.413,A -85,B 0,C 180,E1 -1509.893,E2 -1509.893} C_VEL
LIN {X 0,Y 587.601,Z 395.712,A -85,B 0,C 180,E1 -1512.92,E2 -1512.92} C_VEL
LIN {X 0,Y 587.478,Z 418.698,A -85,B 0,C 180,E1 -1515.991,E2 -1515.991} C_VEL
LIN {X 0,Y 587.407,Z 422.524,A -85,B 0,C 180,E1 -1516.497,E2 -1516.497} C_VEL
LIN {X 0,Y 587.899,Z 426.745,A -85,B 0,C 180,E1 -1516.564,E2 -1516.564} C_VEL
LIN {X 0,Y 587.744,Z 530.961,A -85,B 0,C 180,E1 -1517.856,E2 -1517.856} C_VEL
LIN {X 0,Y 587.668,Z 544.228,A -85,B 0,C 180,E1 -1518.161,E2 -1518.161} C_VEL
LIN {X 0,Y 587.616,Z 556.817,A -85,B 0,C 180,E1 -1518.592,E2 -1518.592} C_VEL
LIN {X 0,Y 587.552,Z 568.636,A -85,B 0,C 180,E1 -1519.141,E2 -1519.141} C_VEL
LIN {X 0,Y 587.465,Z 580.205,A -85,B 0,C 180,E1 -1519.837,E2 -1519.837} C_VEL
LIN {X 0,Y 587.391,Z 590.6,A -85,B 0,C 180,E1 -1520.618,E2 -1520.618} C_VEL
LIN {X 0,Y 587.321,Z 599.114,A -85,B 0,C 180,E1 -1521.398,E2 -1521.398} C_VEL
LIN {X 0,Y 587.273,Z 606.962,A -85,B 0,C 180,E1 -1522.263,E2 -1522.263} C_VEL
LIN {X 0,Y 587.23,Z 613.47,A -85,B 0,C 180,E1 -1523.126,E2 -1523.126} C_VEL
LIN {X 0,Y 587.236,Z 619.867,A -85,B 0,C 180,E1 -1524.161,E2 -1524.161} C_VEL
LIN {X 0,Y 587.147,Z 624.95,A -85,B 0,C 180,E1 -1525.194,E2 -1525.194} C_VEL
LIN {X 0,Y 587.212,Z 628.896,A -85,B 0,C 180,E1 -1526.226,E2 -1526.226} C_VEL
LIN {X 0,Y 587.132,Z 631.809,A -85,B 0,C 180,E1 -1527.256,E2 -1527.256} C_VEL
LIN {X 0,Y 587.139,Z 633.2,A -85,B 0,C 180,E1 -1527.942,E2 -1527.942} C_VEL
LIN {X 0,Y 587.14,Z 634.784,A -85,B 0,C 180,E1 -1529.314,E2 -1529.314} C_VEL
LIN {X 0,Y 587.137,Z 635,A -85,B 0,C 180,E1 -1530,E2 -1530} C_VEL
LIN {X 0,Y 587.147,Z 634.185,A -85,B 0,C 180,E1 -1531.372,E2 -1531.372} C_VEL
LIN {X 0,Y 587.139,Z 633.201,A -85,B 0,C 180,E1 -1532.058,E2 -1532.058} C_VEL
LIN {X 0,Y 587.132,Z 631.81,A -85,B 0,C 180,E1 -1532.744,E2 -1532.744} C_VEL
LIN {X 0,Y 587.212,Z 628.896,A -85,B 0,C 180,E1 -1533.774,E2 -1533.774} C_VEL
LIN {X 0,Y 587.147,Z 624.95,A -85,B 0,C 180,E1 -1534.806,E2 -1534.806} C_VEL
LIN {X 0,Y 587.217,Z 618.878,A -85,B 0,C 180,E1 -1536.011,E2 -1536.011} C_VEL
LIN {X 0,Y 587.245,Z 612.238,A -85,B 0,C 180,E1 -1537.046,E2 -1537.046} C_VEL
LIN {X 0,Y 587.299,Z 603.992,A -85,B 0,C 180,E1 -1538.083,E2 -1538.083} C_VEL
LIN {X 0,Y 587.343,Z 595.54,A -85,B 0,C 180,E1 -1538.949,E2 -1538.949} C_VEL
LIN {X 0,Y 587.416,Z 585.098,A -85,B 0,C 180,E1 -1539.816,E2 -1539.816} C_VEL
LIN {X 0,Y 587.496,Z 574.762,A -85,B 0,C 180,E1 -1540.511,E2 -1540.511} C_VEL
LIN {X 0,Y 587.583,Z 562.811,A -85,B 0,C 180,E1 -1541.149,E2 -1541.149} C_VEL
LIN {X 0,Y 587.624,Z 550.601,A -85,B 0,C 180,E1 -1541.639,E2 -1541.639} C_VEL
LIN {X 0,Y 587.696,Z 537.447,A -85,B 0,C 180,E1 -1542.014,E2 -1542.014} C_VEL
LIN {X 0,Y 587.775,Z 525.105,A -85,B 0,C 180,E1 -1542.231,E2 -1542.231} C_VEL
LIN {X 0,Y 587.731,Z 424.509,A -85,B 0,C 180,E1 -1543.467,E2 -1543.467} C_VEL
LIN {X 0,Y 587.409,Z 422.441,A -85,B 0,C 180,E1 -1543.513,E2 -1543.513} C_VEL
LIN {X 0,Y 587.554,Z 401.334,A -85,B 0,C 180,E1 -1546.325,E2 -1546.325} C_VEL
LIN {X 0,Y 587.736,Z 378.407,A -85,B 0,C 180,E1 -1549.424,E2 -1549.424} C_VEL
LIN {X 0,Y 587.899,Z 356.128,A -85,B 0,C 180,E1 -1552.491,E2 -1552.491} C_VEL
LIN {X 0,Y 587.824,Z 350.81,A -85,B 0,C 180,E1 -1553.237,E2 -1553.237} C_VEL
LIN {X 0,Y 587.347,Z 348.324,A -85,B 0,C 180,E1 -1553.631,E2 -1553.631} C_VEL
LIN {X 0,Y 587.341,Z 348.327,A -85,B 0,C 180,E1 -1556.278,E2 -1556.278} C_VEL
LIN {X 0,Y 587.351,Z 348.317,A -85,B 0,C 180,E1 -1559.133,E2 -1559.133} C_VEL
LIN {X 0,Y 587.355,Z 348.322,A -85,B 0,C 180,E1 -1561.837,E2 -1561.837} C_VEL
LIN {X 0,Y 587.357,Z 348.321,A -85,B 0,C 180,E1 -1564.349,E2 -1564.349} C_VEL
LIN {X 0,Y 587.351,Z 348.317,A -85,B 0,C 180,E1 -1566.746,E2 -1566.746} C_VEL
LIN {X 0,Y 587.345,Z 348.318,A -85,B 0,C 180,E1 -1569.358,E2 -1569.358} C_VEL
LIN {X 0,Y 587.331,Z 348.326,A -85,B 0,C 180,E1 -1572.107,E2 -1572.107} C_VEL
LIN {X 0,Y 587.311,Z 348.321,A -85,B 0,C 180,E1 -1574.91,E2 -1574.91} C_VEL
LIN {X 0,Y 587.319,Z 348.32,A -85,B 0,C 180,E1 -1576.994,E2 -1576.994} C_VEL
LIN {X 0,Y 587.324,Z 348.328,A -85,B 0,C 180,E1 -1579.746,E2 -1579.746} C_VEL
LIN {X 0,Y 587.342,Z 348.319,A -85,B 0,C 180,E1 -1582.392,E2 -1582.392} C_VEL
LIN {X 0,Y 587.341,Z 348.318,A -85,B 0,C 180,E1 -1584.945,E2 -1584.945} C_VEL
LIN {X 0,Y 587.335,Z 348.322,A -85,B 0,C 180,E1 -1587.421,E2 -1587.421} C_VEL
LIN {X 0,Y 587.339,Z 348.326,A -85,B 0,C 180,E1 -1589.83,E2 -1589.83} C_VEL
LIN {X 0,Y 587.343,Z 348.319,A -85,B 0,C 180,E1 -1592.306,E2 -1592.306} C_VEL
LIN {X 0,Y 587.33,Z 348.319,A -85,B 0,C 180,E1 -1594.483,E2 -1594.483} C_VEL
LIN {X 0,Y 587.334,Z 348.326,A -85,B 0,C 180,E1 -1597.486,E2 -1597.486} C_VEL
LIN {X 0,Y 587.327,Z 348.328,A -85,B 0,C 180,E1 -1599.695,E2 -1599.695} C_VEL
LIN {X 0,Y 587.352,Z 348.315,A -85,B 0,C 180,E1 -1602.594,E2 -1602.594} C_VEL
LIN {X 0,Y 587.355,Z 348.322,A -85,B 0,C 180,E1 -1605.739,E2 -1605.739} C_VEL
LIN {X 0,Y 587.352,Z 348.317,A -85,B 0,C 180,E1 -1608.859,E2 -1608.859} C_VEL
LIN {X 0,Y 587.364,Z 348.319,A -85,B 0,C 180,E1 -1611.745,E2 -1611.745} C_VEL
LIN {X 0,Y 587.354,Z 348.316,A -85,B 0,C 180,E1 -1614.507,E2 -1614.507} C_VEL
LIN {X 0,Y 587.377,Z 348.321,A -85,B 0,C 180,E1 -1617.257,E2 -1617.257} C_VEL
LIN {X 0,Y 587.373,Z 348.315,A -85,B 0,C 180,E1 -1620,E2 -1620} C_VEL
LIN {X 0,Y 587.376,Z 348.314,A -85,B 0,C 180,E1 -1622.743,E2 -1622.743} C_VEL
LIN {X 0,Y 587.359,Z 348.321,A -85,B 0,C 180,E1 -1625.493,E2 -1625.493} C_VEL
LIN {X 0,Y 587.364,Z 348.314,A -85,B 0,C 180,E1 -1628.256,E2 -1628.256} C_VEL
LIN {X 0,Y 587.353,Z 348.326,A -85,B 0,C 180,E1 -1631.142,E2 -1631.142} C_VEL
LIN {X 0,Y 587.356,Z 348.316,A -85,B 0,C 180,E1 -1634.262,E2 -1634.262} C_VEL
LIN {X 0,Y 587.354,Z 348.321,A -85,B 0,C 180,E1 -1637.406,E2 -1637.406} C_VEL
LIN {X 0,Y 587.322,Z 348.32,A -85,B 0,C 180,E1 -1638.327,E2 -1638.327} C_VEL
LIN {X 0,Y 586.667,Z 348.409,A -85,B 0,C 180,E1 -1638.899,E2 -1638.899} C_VEL
LIN {X 0,Y 583.832,Z 348.766,A -85,B 0,C 180,E1 -1639.828,E2 -1639.828} C_VEL
LIN {X 0,Y 581.423,Z 349.067,A -85,B 0,C 180,E1 -1640.575,E2 -1640.575} C_VEL
LIN {X 0,Y 580.375,Z 349.194,A -85,B 0,C 180,E1 -1641.151,E2 -1641.151} C_VEL
LIN {X 0,Y 580.283,Z 349.202,A -85,B 0,C 180,E1 -1641.346,E2 -1641.346} C_VEL
LIN {X 0,Y 580.295,Z 349.197,A -85,B 0,C 180,E1 -1643.558,E2 -1643.558} C_VEL
LIN {X 0,Y 580.322,Z 349.193,A -85,B 0,C 180,E1 -1646.343,E2 -1646.343} C_VEL
LIN {X 0,Y 580.299,Z 349.199,A -85,B 0,C 180,E1 -1649.311,E2 -1649.311} C_VEL
LIN {X 0,Y 580.3,Z 349.196,A -85,B 0,C 180,E1 -1652.201,E2 -1652.201} C_VEL
LIN {X 0,Y 580.298,Z 349.201,A -85,B 0,C 180,E1 -1654.696,E2 -1654.696} C_VEL
LIN {X 0,Y 580.297,Z 349.198,A -85,B 0,C 180,E1 -1657.269,E2 -1657.269} C_VEL
LIN {X 0,Y 580.296,Z 349.197,A -85,B 0,C 180,E1 -1660.273,E2 -1660.273} C_VEL
LIN {X 0,Y 580.289,Z 349.205,A -85,B 0,C 180,E1 -1662.706,E2 -1662.706} C_VEL
LIN {X 0,Y 580.272,Z 349.198,A -85,B 0,C 180,E1 -1665.61,E2 -1665.61} C_VEL
LIN {X 0,Y 580.313,Z 349.196,A -85,B 0,C 180,E1 -1668.235,E2 -1668.235} C_VEL
LIN {X 0,Y 580.291,Z 349.202,A -85,B 0,C 180,E1 -1670.967,E2 -1670.967} C_VEL
LIN {X 0,Y 580.297,Z 349.197,A -85,B 0,C 180,E1 -1673.599,E2 -1673.599} C_VEL
LIN {X 0,Y 580.327,Z 349.317,A -85,B 0,C 180,E1 -1675.728,E2 -1675.728} C_VEL
LIN {X 0,Y 580.395,Z 360.496,A -85,B 0,C 180,E1 -1677.806,E2 -1677.806} C_VEL
LIN {X 0,Y 580.273,Z 374.61,A -85,B 0,C 180,E1 -1680.394,E2 -1680.394} C_VEL
LIN {X 0,Y 580.965,Z 380.78,A -85,B 0,C 180,E1 -1680.496,E2 -1680.496} C_VEL
LIN {X 0,Y 580.815,Z 481.735,A -85,B 0,C 180,E1 -1681.769,E2 -1681.769} C_VEL
LIN {X 0,Y 580.707,Z 495.097,A -85,B 0,C 180,E1 -1682.087,E2 -1682.087} C_VEL
LIN {X 0,Y 580.637,Z 507.781,A -85,B 0,C 180,E1 -1682.537,E2 -1682.537} C_VEL
LIN {X 0,Y 580.543,Z 519.453,A -85,B 0,C 180,E1 -1683.099,E2 -1683.099} C_VEL
LIN {X 0,Y 580.445,Z 531.504,A -85,B 0,C 180,E1 -1683.847,E2 -1683.847} C_VEL
LIN {X 0,Y 580.367,Z 541.646,A -85,B 0,C 180,E1 -1684.636,E2 -1684.636} C_VEL
LIN {X 0,Y 580.29,Z 550.509,A -85,B 0,C 180,E1 -1685.483,E2 -1685.483} C_VEL
LIN {X 0,Y 580.198,Z 558.731,A -85,B 0,C 180,E1 -1686.439,E2 -1686.439} C_VEL
LIN {X 0,Y 580.154,Z 566.581,A -85,B 0,C 180,E1 -1687.568,E2 -1687.568} C_VEL
LIN {X 0,Y 580.113,Z 572.702,A -85,B 0,C 180,E1 -1688.689,E2 -1688.689} C_VEL
LIN {X 0,Y 580.091,Z 577.41,A -85,B 0,C 180,E1 -1689.801,E2 -1689.801} C_VEL
LIN {X 0,Y 580.07,Z 580.917,A -85,B 0,C 180,E1 -1690.916,E2 -1690.916} C_VEL
LIN {X 0,Y 580.039,Z 582.59,A -85,B 0,C 180,E1 -1691.638,E2 -1691.638} C_VEL
LIN {X 0,Y 580.043,Z 583.844,A -85,B 0,C 180,E1 -1692.368,E2 -1692.368} C_VEL
LIN {X 0,Y 580.043,Z 584.668,A -85,B 0,C 180,E1 -1693.176,E2 -1693.176} C_VEL
LIN {X 0,Y 580.021,Z 584.894,A -85,B 0,C 180,E1 -1694.54,E2 -1694.54} C_VEL
LIN {X 0,Y 580.053,Z 583.776,A -85,B 0,C 180,E1 -1695.766,E2 -1695.766} C_VEL
LIN {X 0,Y 580.063,Z 582.093,A -85,B 0,C 180,E1 -1696.691,E2 -1696.691} C_VEL
LIN {X 0,Y 580.076,Z 579.222,A -85,B 0,C 180,E1 -1697.759,E2 -1697.759} C_VEL
LIN {X 0,Y 580.08,Z 574.895,A -85,B 0,C 180,E1 -1698.923,E2 -1698.923} C_VEL
LIN {X 0,Y 580.133,Z 570.243,A -85,B 0,C 180,E1 -1699.883,E2 -1699.883} C_VEL
LIN {X 0,Y 580.153,Z 563.903,A -85,B 0,C 180,E1 -1700.939,E2 -1700.939} C_VEL
LIN {X 0,Y 580.243,Z 555.973,A -85,B 0,C 180,E1 -1701.993,E2 -1701.993} C_VEL
LIN {X 0,Y 580.303,Z 546.157,A -85,B 0,C 180,E1 -1703.044,E2 -1703.044} C_VEL
LIN {X 0,Y 580.372,Z 535.94,A -85,B 0,C 180,E1 -1703.918,E2 -1703.918} C_VEL
LIN {X 0,Y 580.478,Z 524.46,A -85,B 0,C 180,E1 -1704.703,E2 -1704.703} C_VEL
LIN {X 0,Y 580.61,Z 513.146,A -85,B 0,C 180,E1 -1705.314,E2 -1705.314} C_VEL
LIN {X 0,Y 580.68,Z 500.305,A -85,B 0,C 180,E1 -1705.836,E2 -1705.836} C_VEL
LIN {X 0,Y 580.745,Z 487.427,A -85,B 0,C 180,E1 -1706.205,E2 -1706.205} C_VEL
LIN {X 0,Y 580.814,Z 473.545,A -85,B 0,C 180,E1 -1706.445,E2 -1706.445} C_VEL
LIN {X 0,Y 580.872,Z 378.301,A -85,B 0,C 180,E1 -1707.627,E2 -1707.627} C_VEL
LIN {X 0,Y 580.321,Z 374.578,A -85,B 0,C 180,E1 -1707.701,E2 -1707.701} C_VEL
LIN {X 0,Y 580.434,Z 358.272,A -85,B 0,C 180,E1 -1710.694,E2 -1710.694} C_VEL
LIN {X 0,Y 580.322,Z 349.196,A -85,B 0,C 180,E1 -1712.386,E2 -1712.386} C_VEL
LIN {X 0,Y 580.33,Z 349.2,A -85,B 0,C 180,E1 -1715.56,E2 -1715.56} C_VEL
LIN {X 0,Y 580.317,Z 349.193,A -85,B 0,C 180,E1 -1718.356,E2 -1718.356} C_VEL
LIN {X 0,Y 580.307,Z 349.2,A -85,B 0,C 180,E1 -1721.191,E2 -1721.191} C_VEL
LIN {X 0,Y 580.333,Z 349.192,A -85,B 0,C 180,E1 -1724.016,E2 -1724.016} C_VEL
LIN {X 0,Y 580.318,Z 349.196,A -85,B 0,C 180,E1 -1726.913,E2 -1726.913} C_VEL
LIN {X 0,Y 580.292,Z 349.198,A -85,B 0,C 180,E1 -1729.822,E2 -1729.822} C_VEL
LIN {X 0,Y 580.275,Z 349.198,A -85,B 0,C 180,E1 -1732.052,E2 -1732.052} C_VEL
LIN {X 0,Y 580.311,Z 349.2,A -85,B 0,C 180,E1 -1735.079,E2 -1735.079} C_VEL
LIN {X 0,Y 580.301,Z 349.194,A -85,B 0,C 180,E1 -1738.185,E2 -1738.185} C_VEL
LIN {X 0,Y 580.295,Z 349.198,A -85,B 0,C 180,E1 -1740.695,E2 -1740.695} C_VEL
LIN {X 0,Y 580.305,Z 349.201,A -85,B 0,C 180,E1 -1743.316,E2 -1743.316} C_VEL
LIN {X 0,Y 580.328,Z 349.192,A -85,B 0,C 180,E1 -1745.767,E2 -1745.767} C_VEL
LIN {X 0,Y 580.289,Z 349.196,A -85,B 0,C 180,E1 -1748.145,E2 -1748.145} C_VEL
LIN {X 0,Y 580.299,Z 349.201,A -85,B 0,C 180,E1 -1750.842,E2 -1750.842} C_VEL
LIN {X 0,Y 580.286,Z 349.198,A -85,B 0,C 180,E1 -1753.656,E2 -1753.656} C_VEL
LIN {X 0,Y 580.29,Z 349.199,A -85,B 0,C 180,E1 -1756.607,E2 -1756.607} C_VEL
LIN {X 0,Y 580.299,Z 349.202,A -85,B 0,C 180,E1 -1759.156,E2 -1759.156} C_VEL
LIN {X 0,Y 580.287,Z 349.196,A -85,B 0,C 180,E1 -1761.926,E2 -1761.926} C_VEL
LIN {X 0,Y 580.301,Z 349.197,A -85,B 0,C 180,E1 -1764.456,E2 -1764.456} C_VEL
LIN {X 0,Y 580.288,Z 349.205,A -85,B 0,C 180,E1 -1766.975,E2 -1766.975} C_VEL
LIN {X 0,Y 580.297,Z 349.197,A -85,B 0,C 180,E1 -1769.425,E2 -1769.425} C_VEL
LIN {X 0,Y 580.314,Z 349.194,A -85,B 0,C 180,E1 -1772.136,E2 -1772.136} C_VEL
LIN {X 0,Y 580.302,Z 349.203,A -85,B 0,C 180,E1 -1774.92,E2 -1774.92} C_VEL
LIN {X 0,Y 580.271,Z 349.198,A -85,B 0,C 180,E1 -1777.947,E2 -1777.947} C_VEL
LIN {X 0,Y 580.31,Z 349.2,A -85,B 0,C 180,E1 -1780.913,E2 -1780.913} C_VEL
LIN {X 0,Y 580.277,Z 349.197,A -85,B 0,C 180,E1 -1783.825,E2 -1783.825} C_VEL
LIN {X 0,Y 580.274,Z 349.208,A -85,B 0,C 180,E1 -1786.696,E2 -1786.696} C_VEL
LIN {X 0,Y 580.297,Z 349.195,A -85,B 0,C 180,E1 -1789.533,E2 -1789.533} C_VEL
LIN {X 0,Y 580.324,Z 349.197,A -85,B 0,C 180,E1 -1792.344,E2 -1792.344} C_VEL
LIN {X 0,Y 580.335,Z 349.192,A -85,B 0,C 180,E1 -1795.137,E2 -1795.137} C_VEL
LIN {X 0,Y 580.329,Z 349.192,A -85,B 0,C 180,E1 -1797.918,E2 -1797.918} C_VEL
LIN {X 0,Y 580.359,Z 349.194,A -85,B 0,C 180,E1 -1800.694,E2 -1800.694} C_VEL
LIN {X 0,Y 580.282,Z 349.197,A -85,B 0,C 180,E1 -1803.472,E2 -1803.472} C_VEL
LIN {X 0,Y 580.317,Z 349.192,A -85,B 0,C 180,E1 -1805.56,E2 -1805.56} C_VEL
LIN {X 0,Y 580.326,Z 349.2,A -85,B 0,C 180,E1 -1808.356,E2 -1808.356} C_VEL
LIN {X 0,Y 580.323,Z 349.192,A -85,B 0,C 180,E1 -1811.208,E2 -1811.208} C_VEL
LIN {X 0,Y 580.305,Z 349.204,A -85,B 0,C 180,E1 -1814.339,E2 -1814.339} C_VEL
LIN {X 0,Y 580.307,Z 349.195,A -85,B 0,C 180,E1 -1816.916,E2 -1816.916} C_VEL
LIN {X 0,Y 580.3,Z 349.197,A -85,B 0,C 180,E1 -1819.822,E2 -1819.822} C_VEL
LIN {X 0,Y 580.272,Z 349.204,A -85,B 0,C 180,E1 -1822.053,E2 -1822.053} C_VEL
LIN {X 0,Y 580.3,Z 349.195,A -85,B 0,C 180,E1 -1825.08,E2 -1825.08} C_VEL
LIN {X 0,Y 580.312,Z 349.197,A -85,B 0,C 180,E1 -1827.864,E2 -1827.864} C_VEL
LIN {X 0,Y 580.292,Z 349.198,A -85,B 0,C 180,E1 -1830.698,E2 -1830.698} C_VEL
LIN {X 0,Y 580.3,Z 349.195,A -85,B 0,C 180,E1 -1833.318,E2 -1833.318} C_VEL
LIN {X 0,Y 580.319,Z 349.196,A -85,B 0,C 180,E1 -1835.768,E2 -1835.768} C_VEL
LIN {X 0,Y 580.285,Z 349.206,A -85,B 0,C 180,E1 -1838.147,E2 -1838.147} C_VEL
LIN {X 0,Y 580.301,Z 349.195,A -85,B 0,C 180,E1 -1840.843,E2 -1840.843} C_VEL
LIN {X 0,Y 580.284,Z 349.2,A -85,B 0,C 180,E1 -1843.657,E2 -1843.657} C_VEL
LIN {X 0,Y 580.281,Z 349.198,A -85,B 0,C 180,E1 -1846.609,E2 -1846.609} C_VEL
LIN {X 0,Y 580.302,Z 349.194,A -85,B 0,C 180,E1 -1849.158,E2 -1849.158} C_VEL
LIN {X 0,Y 580.289,Z 349.206,A -85,B 0,C 180,E1 -1851.927,E2 -1851.927} C_VEL
LIN {X 0,Y 580.307,Z 349.196,A -85,B 0,C 180,E1 -1854.458,E2 -1854.458} C_VEL
LIN {X 0,Y 580.291,Z 349.196,A -85,B 0,C 180,E1 -1856.976,E2 -1856.976} C_VEL
LIN {X 0,Y 580.311,Z 349.196,A -85,B 0,C 180,E1 -1859.427,E2 -1859.427} C_VEL
LIN {X 0,Y 580.321,Z 349.199,A -85,B 0,C 180,E1 -1862.138,E2 -1862.138} C_VEL
LIN {X 0,Y 580.323,Z 349.196,A -85,B 0,C 180,E1 -1865.27,E2 -1865.27} C_VEL
LIN {X 0,Y 580.312,Z 349.314,A -85,B 0,C 180,E1 -1866.231,E2 -1866.231} C_VEL
LIN {X 0,Y 581.032,Z 354.158,A -85,B 0,C 180,E1 -1866.95,E2 -1866.95} C_VEL
LIN {X 0,Y 580.837,Z 373.413,A -85,B 0,C 180,E1 -1869.644,E2 -1869.644} C_VEL
LIN {X 0,Y 580.615,Z 394.819,A -85,B 0,C 180,E1 -1872.586,E2 -1872.586} C_VEL
LIN {X 0,Y 580.467,Z 416.36,A -85,B 0,C 180,E1 -1875.504,E2 -1875.504} C_VEL
LIN {X 0,Y 580.415,Z 422.524,A -85,B 0,C 180,E1 -1876.332,E2 -1876.332} C_VEL
LIN {X 0,Y 580.983,Z 428.534,A -85,B 0,C 180,E1 -1876.423,E2 -1876.423} C_VEL
LIN {X 0,Y 580.815,Z 530.961,A -85,B 0,C 180,E1 -1877.709,E2 -1877.709} C_VEL
LIN {X 0,Y 580.726,Z 544.229,A -85,B 0,C 180,E1 -1878.017,E2 -1878.017} C_VEL
LIN {X 0,Y 580.664,Z 556.38,A -85,B 0,C 180,E1 -1878.437,E2 -1878.437} C_VEL
LIN {X 0,Y 580.574,Z 568.634,A -85,B 0,C 180,E1 -1879.009,E2 -1879.009} C_VEL
LIN {X 0,Y 580.444,Z 580.206,A -85,B 0,C 180,E1 -1879.712,E2 -1879.712} C_VEL
LIN {X 0,Y 580.341,Z 590.602,A -85,B 0,C 180,E1 -1880.503,E2 -1880.503} C_VEL
LIN {X 0,Y 580.271,Z 599.114,A -85,B 0,C 180,E1 -1881.292,E2 -1881.292} C_VEL
LIN {X 0,Y 580.221,Z 606.962,A -85,B 0,C 180,E1 -1882.168,E2 -1882.168} C_VEL
LIN {X 0,Y 580.153,Z 614.651,A -85,B 0,C 180,E1 -1883.222,E2 -1883.222} C_VEL
LIN {X 0,Y 580.139,Z 621.681,A -85,B 0,C 180,E1 -1884.439,E2 -1884.439} C_VEL
LIN {X 0,Y 580.108,Z 626.372,A -85,B 0,C 180,E1 -1885.484,E2 -1885.484} C_VEL
LIN {X 0,Y 580.123,Z 629.957,A -85,B 0,C 180,E1 -1886.527,E2 -1886.527} C_VEL
LIN {X 0,Y 580.043,Z 631.809,A -85,B 0,C 180,E1 -1887.222,E2 -1887.222} C_VEL
LIN {X 0,Y 580.038,Z 633.199,A -85,B 0,C 180,E1 -1887.917,E2 -1887.917} C_VEL
LIN {X 0,Y 580.04,Z 634.785,A -85,B 0,C 180,E1 -1889.306,E2 -1889.306} C_VEL
LIN {X 0,Y 580.037,Z 635,A -85,B 0,C 180,E1 -1890,E2 -1890} C_VEL
LIN {X 0,Y 580.047,Z 634.186,A -85,B 0,C 180,E1 -1891.389,E2 -1891.389} C_VEL
LIN {X 0,Y 580.038,Z 633.2,A -85,B 0,C 180,E1 -1892.083,E2 -1892.083} C_VEL
LIN {X 0,Y 580.043,Z 631.81,A -85,B 0,C 180,E1 -1892.778,E2 -1892.778} C_VEL
LIN {X 0,Y 580.109,Z 628.896,A -85,B 0,C 180,E1 -1893.82,E2 -1893.82} C_VEL
LIN {X 0,Y 580.054,Z 624.95,A -85,B 0,C 180,E1 -1894.865,E2 -1894.865} C_VEL
LIN {X 0,Y 580.139,Z 618.878,A -85,B 0,C 180,E1 -1896.085,E2 -1896.085} C_VEL
LIN {X 0,Y 580.184,Z 612.238,A -85,B 0,C 180,E1 -1897.132,E2 -1897.132} C_VEL
LIN {X 0,Y 580.25,Z 603.992,A -85,B 0,C 180,E1 -1898.182,E2 -1898.182} C_VEL
LIN {X 0,Y 580.308,Z 595.54,A -85,B 0,C 180,E1 -1899.058,E2 -1899.058} C_VEL
LIN {X 0,Y 580.417,Z 585.1,A -85,B 0,C 180,E1 -1899.936,E2 -1899.936} C_VEL
LIN {X 0,Y 580.507,Z 574.76,A -85,B 0,C 180,E1 -1900.639,E2 -1900.639} C_VEL
LIN {X 0,Y 580.596,Z 563.241,A -85,B 0,C 180,E1 -1901.264,E2 -1901.264} C_VEL
LIN {X 0,Y 580.664,Z 550.479,A -85,B 0,C 180,E1 -1901.785,E2 -1901.785} C_VEL
LIN {X 0,Y 580.743,Z 537.446,A -85,B 0,C 180,E1 -1902.16,E2 -1902.16} C_VEL
LIN {X 0,Y 580.859,Z 525.105,A -85,B 0,C 180,E1 -1902.379,E2 -1902.379} C_VEL
LIN {X 0,Y 580.815,Z 425.182,A -85,B 0,C 180,E1 -1903.622,E2 -1903.622} C_VEL
LIN {X 0,Y 580.419,Z 422.441,A -85,B 0,C 180,E1 -1903.679,E2 -1903.679} C_VEL
LIN {X 0,Y 580.571,Z 400.004,A -85,B 0,C 180,E1 -1906.708,E2 -1906.708} C_VEL
LIN {X 0,Y 580.793,Z 377.402,A -85,B 0,C 180,E1 -1909.804,E2 -1909.804} C_VEL
LIN {X 0,Y 581.038,Z 356.128,A -85,B 0,C 180,E1 -1912.771,E2 -1912.771} C_VEL
LIN {X 0,Y 580.952,Z 352.486,A -85,B 0,C 180,E1 -1913.29,E2 -1913.29} C_VEL
LIN {X 0,Y 580.302,Z 349.203,A -85,B 0,C 180,E1 -1913.793,E2 -1913.793} C_VEL
LIN {X 0,Y 580.278,Z 349.202,A -85,B 0,C 180,E1 -1916.623,E2 -1916.623} C_VEL
LIN {X 0,Y 580.306,Z 349.195,A -85,B 0,C 180,E1 -1919.31,E2 -1919.31} C_VEL
LIN {X 0,Y 580.302,Z 349.203,A -85,B 0,C 180,E1 -1922.199,E2 -1922.199} C_VEL
LIN {X 0,Y 580.301,Z 349.196,A -85,B 0,C 180,E1 -1924.695,E2 -1924.695} C_VEL
LIN {X 0,Y 580.298,Z 349.196,A -85,B 0,C 180,E1 -1927.267,E2 -1927.267} C_VEL
LIN {X 0,Y 580.304,Z 349.2,A -85,B 0,C 180,E1 -1930.272,E2 -1930.272} C_VEL
LIN {X 0,Y 580.277,Z 349.198,A -85,B 0,C 180,E1 -1932.705,E2 -1932.705} C_VEL
LIN {X 0,Y 580.27,Z 349.203,A -85,B 0,C 180,E1 -1935.608,E2 -1935.608} C_VEL
LIN {X 0,Y 580.31,Z 349.198,A -85,B 0,C 180,E1 -1938.234,E2 -1938.234} C_VEL
LIN {X 0,Y 580.285,Z 349.196,A -85,B 0,C 180,E1 -1940.966,E2 -1940.966} C_VEL
LIN {X 0,Y 580.29,Z 349.202,A -85,B 0,C 180,E1 -1943.598,E2 -1943.598} C_VEL
LIN {X 0,Y 580.313,Z 349.197,A -85,B 0,C 180,E1 -1946.145,E2 -1946.145} C_VEL
LIN {X 0,Y 580.284,Z 349.197,A -85,B 0,C 180,E1 -1948.615,E2 -1948.615} C_VEL
LIN {X 0,Y 580.288,Z 349.197,A -85,B 0,C 180,E1 -1951.024,E2 -1951.024} C_VEL
LIN {X 0,Y 580.32,Z 349.201,A -85,B 0,C 180,E1 -1953.658,E2 -1953.658} C_VEL
LIN {X 0,Y 580.271,Z 349.198,A -85,B 0,C 180,E1 -1956.442,E2 -1956.442} C_VEL
LIN {X 0,Y 580.276,Z 349.204,A -85,B 0,C 180,E1 -1959.437,E2 -1959.437} C_VEL
LIN {X 0,Y 580.275,Z 349.206,A -85,B 0,C 180,E1 -1961.645,E2 -1961.645} C_VEL
LIN {X 0,Y 580.276,Z 349.203,A -85,B 0,C 180,E1 -1963.826,E2 -1963.826} C_VEL
LIN {X 0,Y 580.271,Z 349.198,A -85,B 0,C 180,E1 -1966.696,E2 -1966.696} C_VEL
LIN {X 0,Y 580.296,Z 349.204,A -85,B 0,C 180,E1 -1969.533,E2 -1969.533} C_VEL
LIN {X 0,Y 580.324,Z 349.19,A -85,B 0,C 180,E1 -1972.345,E2 -1972.345} C_VEL
LIN {X 0,Y 580.338,Z 349.196,A -85,B 0,C 180,E1 -1975.137,E2 -1975.137} C_VEL
LIN {X 0,Y 580.33,Z 349.192,A -85,B 0,C 180,E1 -1977.918,E2 -1977.918} C_VEL
LIN {X 0,Y 580.361,Z 349.188,A -85,B 0,C 180,E1 -1980.694,E2 -1980.694} C_VEL
LIN {X 0,Y 580.287,Z 349.203,A -85,B 0,C 180,E1 -1983.472,E2 -1983.472} C_VEL
LIN {X 0,Y 580.323,Z 349.197,A -85,B 0,C 180,E1 -1985.56,E2 -1985.56} C_VEL
LIN {X 0,Y 580.328,Z 349.191,A -85,B 0,C 180,E1 -1988.356,E2 -1988.356} C_VEL
LIN {X 0,Y 580.324,Z 349.201,A -85,B 0,C 180,E1 -1991.209,E2 -1991.209} C_VEL
LIN {X 0,Y 580.319,Z 349.192,A -85,B 0,C 180,E1 -1994.017,E2 -1994.017} C_VEL
LIN {X 0,Y 580.308,Z 349.2,A -85,B 0,C 180,E1 -1996.916,E2 -1996.916} C_VEL
LIN {X 0,Y 580.302,Z 349.194,A -85,B 0,C 180,E1 -1999.823,E2 -1999.823} C_VEL
LIN {X 0,Y 580.283,Z 349.202,A -85,B 0,C 180,E1 -2001.346,E2 -2001.346} C_VEL
LIN {X 0,Y 579.593,Z 349.285,A -85,B 0,C 180,E1 -2001.926,E2 -2001.926} C_VEL
LIN {X 0,Y 576.72,Z 349.648,A -85,B 0,C 180,E1 -2002.866,E2 -2002.866} C_VEL
LIN {X 0,Y 574.322,Z 349.942,A -85,B 0,C 180,E1 -2003.622,E2 -2003.622} C_VEL
LIN {X 0,Y 573.317,Z 350.064,A -85,B 0,C 180,E1 -2004.206,E2 -2004.206} C_VEL
LIN {X 0,Y 573.248,Z 350.074,A -85,B 0,C 180,E1 -2004.404,E2 -2004.404} C_VEL
LIN {X 0,Y 573.262,Z 350.081,A -85,B 0,C 180,E1 -2006.976,E2 -2006.976} C_VEL
LIN {X 0,Y 573.244,Z 350.076,A -85,B 0,C 180,E1 -2009.49,E2 -2009.49} C_VEL
LIN {X 0,Y 573.253,Z 350.074,A -85,B 0,C 180,E1 -2012.23,E2 -2012.23} C_VEL
LIN {X 0,Y 573.248,Z 350.08,A -85,B 0,C 180,E1 -2014.775,E2 -2014.775} C_VEL
LIN {X 0,Y 573.251,Z 350.077,A -85,B 0,C 180,E1 -2017.167,E2 -2017.167} C_VEL
LIN {X 0,Y 573.245,Z 350.074,A -85,B 0,C 180,E1 -2019.608,E2 -2019.608} C_VEL
LIN {X 0,Y 573.249,Z 350.081,A -85,B 0,C 180,E1 -2022.644,E2 -2022.644} C_VEL
LIN {X 0,Y 573.237,Z 350.075,A -85,B 0,C 180,E1 -2025.668,E2 -2025.668} C_VEL
LIN {X 0,Y 573.244,Z 350.081,A -85,B 0,C 180,E1 -2028.545,E2 -2028.545} C_VEL
LIN {X 0,Y 573.25,Z 350.076,A -85,B 0,C 180,E1 -2031.3,E2 -2031.3} C_VEL
LIN {X 0,Y 573.266,Z 350.075,A -85,B 0,C 180,E1 -2034.012,E2 -2034.012} C_VEL
LIN {X 0,Y 573.32,Z 350.267,A -85,B 0,C 180,E1 -2035.676,E2 -2035.676} C_VEL
LIN {X 0,Y 573.378,Z 361.302,A -85,B 0,C 180,E1 -2037.753,E2 -2037.753} C_VEL
LIN {X 0,Y 573.274,Z 374.595,A -85,B 0,C 180,E1 -2040.221,E2 -2040.221} C_VEL
LIN {X 0,Y 574.075,Z 381.384,A -85,B 0,C 180,E1 -2040.338,E2 -2040.338} C_VEL
LIN {X 0,Y 573.878,Z 481.373,A -85,B 0,C 180,E1 -2041.611,E2 -2041.611} C_VEL
LIN {X 0,Y 573.767,Z 494.836,A -85,B 0,C 180,E1 -2041.933,E2 -2041.933} C_VEL
LIN {X 0,Y 573.7,Z 506.808,A -85,B 0,C 180,E1 -2042.356,E2 -2042.356} C_VEL
LIN {X 0,Y 573.55,Z 519.052,A -85,B 0,C 180,E1 -2042.941,E2 -2042.941} C_VEL
LIN {X 0,Y 573.445,Z 531.283,A -85,B 0,C 180,E1 -2043.706,E2 -2043.706} C_VEL
LIN {X 0,Y 573.325,Z 541.386,A -85,B 0,C 180,E1 -2044.497,E2 -2044.497} C_VEL
LIN {X 0,Y 573.242,Z 550.401,A -85,B 0,C 180,E1 -2045.365,E2 -2045.365} C_VEL
LIN {X 0,Y 573.139,Z 558.565,A -85,B 0,C 180,E1 -2046.323,E2 -2046.323} C_VEL
LIN {X 0,Y 573.08,Z 566.444,A -85,B 0,C 180,E1 -2047.466,E2 -2047.466} C_VEL
LIN {X 0,Y 573.021,Z 571.667,A -85,B 0,C 180,E1 -2048.412,E2 -2048.412} C_VEL
LIN {X 0,Y 573.006,Z 576.646,A -85,B 0,C 180,E1 -2049.54,E2 -2049.54} C_VEL
LIN {X 0,Y 572.972,Z 580.768,A -85,B 0,C 180,E1 -2050.818,E2 -2050.818} C_VEL
LIN {X 0,Y 572.946,Z 583.527,A -85,B 0,C 180,E1 -2052.142,E2 -2052.142} C_VEL
LIN {X 0,Y 572.942,Z 584.621,A -85,B 0,C 180,E1 -2053.097,E2 -2053.097} C_VEL
LIN {X 0,Y 572.916,Z 584.94,A -85,B 0,C 180,E1 -2054.344,E2 -2054.344} C_VEL
LIN {X 0,Y 572.946,Z 583.888,A -85,B 0,C 180,E1 -2055.709,E2 -2055.709} C_VEL
LIN {X 0,Y 572.972,Z 582.504,A -85,B 0,C 180,E1 -2056.524,E2 -2056.524} C_VEL
LIN {X 0,Y 572.994,Z 579.823,A -85,B 0,C 180,E1 -2057.606,E2 -2057.606} C_VEL
LIN {X 0,Y 572.996,Z 575.3,A -85,B 0,C 180,E1 -2058.884,E2 -2058.884} C_VEL
LIN {X 0,Y 573.043,Z 569.401,A -85,B 0,C 180,E1 -2060.114,E2 -2060.114} C_VEL
LIN {X 0,Y 573.106,Z 562.816,A -85,B 0,C 180,E1 -2061.183,E2 -2061.183} C_VEL
LIN {X 0,Y 573.173,Z 554.661,A -85,B 0,C 180,E1 -2062.249,E2 -2062.249} C_VEL
LIN {X 0,Y 573.296,Z 545.612,A -85,B 0,C 180,E1 -2063.208,E2 -2063.208} C_VEL
LIN {X 0,Y 573.406,Z 535.036,A -85,B 0,C 180,E1 -2064.108,E2 -2064.108} C_VEL
LIN {X 0,Y 573.498,Z 523.363,A -85,B 0,C 180,E1 -2064.903,E2 -2064.903} C_VEL
LIN {X 0,Y 573.661,Z 511.654,A -85,B 0,C 180,E1 -2065.521,E2 -2065.521} C_VEL
LIN {X 0,Y 573.72,Z 499.607,A -85,B 0,C 180,E1 -2066.005,E2 -2066.005} C_VEL
LIN {X 0,Y 573.837,Z 486.391,A -85,B 0,C 180,E1 -2066.379,E2 -2066.379} C_VEL
LIN {X 0,Y 573.887,Z 473.335,A -85,B 0,C 180,E1 -2066.599,E2 -2066.599} C_VEL
LIN {X 0,Y 573.964,Z 378.992,A -85,B 0,C 180,E1 -2067.785,E2 -2067.785} C_VEL
LIN {X 0,Y 573.293,Z 374.584,A -85,B 0,C 180,E1 -2067.87,E2 -2067.87} C_VEL
LIN {X 0,Y 573.419,Z 359.345,A -85,B 0,C 180,E1 -2070.702,E2 -2070.702} C_VEL
LIN {X 0,Y 573.299,Z 350.149,A -85,B 0,C 180,E1 -2072.437,E2 -2072.437} C_VEL
LIN {X 0,Y 573.296,Z 350.075,A -85,B 0,C 180,E1 -2075.628,E2 -2075.628} C_VEL
LIN {X 0,Y 573.261,Z 350.072,A -85,B 0,C 180,E1 -2078.46,E2 -2078.46} C_VEL
LIN {X 0,Y 573.278,Z 350.078,A -85,B 0,C 180,E1 -2081.312,E2 -2081.312} C_VEL
LIN {X 0,Y 573.288,Z 350.068,A -85,B 0,C 180,E1 -2084.424,E2 -2084.424} C_VEL
LIN {X 0,Y 573.264,Z 350.077,A -85,B 0,C 180,E1 -2087.111,E2 -2087.111} C_VEL
LIN {X 0,Y 573.246,Z 350.074,A -85,B 0,C 180,E1 -2090.076,E2 -2090.076} C_VEL
LIN {X 0,Y 573.24,Z 350.074,A -85,B 0,C 180,E1 -2092.337,E2 -2092.337} C_VEL
LIN {X 0,Y 573.259,Z 350.079,A -85,B 0,C 180,E1 -2095.409,E2 -2095.409} C_VEL
LIN {X 0,Y 573.253,Z 350.073,A -85,B 0,C 180,E1 -2098.028,E2 -2098.028} C_VEL
LIN {X 0,Y 573.241,Z 350.079,A -85,B 0,C 180,E1 -2100.883,E2 -2100.883} C_VEL
LIN {X 0,Y 573.263,Z 350.075,A -85,B 0,C 180,E1 -2103.523,E2 -2103.523} C_VEL
LIN {X 0,Y 573.262,Z 350.071,A -85,B 0,C 180,E1 -2106.047,E2 -2106.047} C_VEL
LIN {X 0,Y 573.25,Z 350.076,A -85,B 0,C 180,E1 -2108.7,E2 -2108.7} C_VEL
LIN {X 0,Y 573.252,Z 350.075,A -85,B 0,C 180,E1 -2111.595,E2 -2111.595} C_VEL
LIN {X 0,Y 573.237,Z 350.075,A -85,B 0,C 180,E1 -2114.332,E2 -2114.332} C_VEL
LIN {X 0,Y 573.249,Z 350.077,A -85,B 0,C 180,E1 -2117.356,E2 -2117.356} C_VEL
LIN {X 0,Y 573.245,Z 350.075,A -85,B 0,C 180,E1 -2120.392,E2 -2120.392} C_VEL
LIN {X 0,Y 573.253,Z 350.08,A -85,B 0,C 180,E1 -2123.077,E2 -2123.077} C_VEL
LIN {X 0,Y 573.268,Z 350.071,A -85,B 0,C 180,E1 -2125.671,E2 -2125.671} C_VEL
LIN {X 0,Y 573.246,Z 350.074,A -85,B 0,C 180,E1 -2128.184,E2 -2128.184} C_VEL
LIN {X 0,Y 573.26,Z 350.078,A -85,B 0,C 180,E1 -2130.633,E2 -2130.633} C_VEL
LIN {X 0,Y 573.266,Z 350.072,A -85,B 0,C 180,E1 -2133.499,E2 -2133.499} C_VEL
LIN {X 0,Y 573.226,Z 350.077,A -85,B 0,C 180,E1 -2136.134,E2 -2136.134} C_VEL
LIN {X 0,Y 573.254,Z 350.076,A -85,B 0,C 180,E1 -2139.173,E2 -2139.173} C_VEL
LIN {X 0,Y 573.232,Z 350.076,A -85,B 0,C 180,E1 -2141.411,E2 -2141.411} C_VEL
LIN {X 0,Y 573.252,Z 350.072,A -85,B 0,C 180,E1 -2143.621,E2 -2143.621} C_VEL
LIN {X 0,Y 573.232,Z 350.083,A -85,B 0,C 180,E1 -2146.529,E2 -2146.529} C_VEL
LIN {X 0,Y 573.267,Z 350.071,A -85,B 0,C 180,E1 -2149.403,E2 -2149.403} C_VEL
LIN {X 0,Y 573.275,Z 350.074,A -85,B 0,C 180,E1 -2152.25,E2 -2152.25} C_VEL
LIN {X 0,Y 573.306,Z 350.068,A -85,B 0,C 180,E1 -2155.077,E2 -2155.077} C_VEL
LIN {X 0,Y 573.3,Z 350.068,A -85,B 0,C 180,E1 -2157.892,E2 -2157.892} C_VEL
LIN {X 0,Y 573.329,Z 350.07,A -85,B 0,C 180,E1 -2160.702,E2 -2160.702} C_VEL
LIN {X 0,Y 573.233,Z 350.075,A -85,B 0,C 180,E1 -2163.514,E2 -2163.514} C_VEL
LIN {X 0,Y 573.284,Z 350.069,A -85,B 0,C 180,E1 -2165.628,E2 -2165.628} C_VEL
LIN {X 0,Y 573.298,Z 350.077,A -85,B 0,C 180,E1 -2168.459,E2 -2168.459} C_VEL
LIN {X 0,Y 573.289,Z 350.068,A -85,B 0,C 180,E1 -2171.312,E2 -2171.312} C_VEL
LIN {X 0,Y 573.271,Z 350.079,A -85,B 0,C 180,E1 -2174.425,E2 -2174.425} C_VEL
LIN {X 0,Y 573.252,Z 350.073,A -85,B 0,C 180,E1 -2177.112,E2 -2177.112} C_VEL
LIN {X 0,Y 573.249,Z 350.079,A -85,B 0,C 180,E1 -2180.077,E2 -2180.077} C_VEL
LIN {X 0,Y 573.234,Z 350.084,A -85,B 0,C 180,E1 -2182.338,E2 -2182.338} C_VEL
LIN {X 0,Y 573.248,Z 350.073,A -85,B 0,C 180,E1 -2185.41,E2 -2185.41} C_VEL
LIN {X 0,Y 573.257,Z 350.079,A -85,B 0,C 180,E1 -2188.032,E2 -2188.032} C_VEL
LIN {X 0,Y 573.237,Z 350.075,A -85,B 0,C 180,E1 -2190.886,E2 -2190.886} C_VEL
LIN {X 0,Y 573.281,Z 350.07,A -85,B 0,C 180,E1 -2193.529,E2 -2193.529} C_VEL
LIN {X 0,Y 573.254,Z 350.081,A -85,B 0,C 180,E1 -2196.049,E2 -2196.049} C_VEL
LIN {X 0,Y 573.244,Z 350.075,A -85,B 0,C 180,E1 -2198.701,E2 -2198.701} C_VEL
LIN {X 0,Y 573.25,Z 350.076,A -85,B 0,C 180,E1 -2201.597,E2 -2201.597} C_VEL
LIN {X 0,Y 573.235,Z 350.08,A -85,B 0,C 180,E1 -2204.334,E2 -2204.334} C_VEL
LIN {X 0,Y 573.239,Z 350.075,A -85,B 0,C 180,E1 -2207.359,E2 -2207.359} C_VEL
LIN {X 0,Y 573.248,Z 350.076,A -85,B 0,C 180,E1 -2210.394,E2 -2210.394} C_VEL
LIN {X 0,Y 573.254,Z 350.072,A -85,B 0,C 180,E1 -2213.079,E2 -2213.079} C_VEL
LIN {X 0,Y 573.274,Z 350.076,A -85,B 0,C 180,E1 -2215.673,E2 -2215.673} C_VEL
LIN {X 0,Y 573.249,Z 350.078,A -85,B 0,C 180,E1 -2218.186,E2 -2218.186} C_VEL
LIN {X 0,Y 573.27,Z 350.072,A -85,B 0,C 180,E1 -2220.635,E2 -2220.635} C_VEL
LIN {X 0,Y 573.252,Z 350.075,A -85,B 0,C 180,E1 -2223.025,E2 -2223.025} C_VEL
LIN {X 0,Y 573.265,Z 350.081,A -85,B 0,C 180,E1 -2226.041,E2 -2226.041} C_VEL
LIN {X 0,Y 574.068,Z 354.119,A -85,B 0,C 180,E1 -2226.662,E2 -2226.662} C_VEL
LIN {X 0,Y 573.941,Z 370.903,A -85,B 0,C 180,E1 -2229.034,E2 -2229.034} C_VEL
LIN {X 0,Y 573.677,Z 390.697,A -85,B 0,C 180,E1 -2231.797,E2 -2231.797} C_VEL
LIN {X 0,Y 573.494,Z 409.311,A -85,B 0,C 180,E1 -2234.36,E2 -2234.36} C_VEL
LIN {X 0,Y 573.412,Z 422.524,A -85,B 0,C 180,E1 -2236.161,E2 -2236.161} C_VEL
LIN {X 0,Y 574.089,Z 428.534,A -85,B 0,C 180,E1 -2236.257,E2 -2236.257} C_VEL
LIN {X 0,Y 573.879,Z 530.961,A -85,B 0,C 180,E1 -2237.558,E2 -2237.558} C_VEL
LIN {X 0,Y 573.799,Z 544.229,A -85,B 0,C 180,E1 -2237.87,E2 -2237.87} C_VEL
LIN {X 0,Y 573.713,Z 556.381,A -85,B 0,C 180,E1 -2238.295,E2 -2238.295} C_VEL
LIN {X 0,Y 573.574,Z 567.595,A -85,B 0,C 180,E1 -2238.818,E2 -2238.818} C_VEL
LIN {X 0,Y 573.469,Z 578.914,A -85,B 0,C 180,E1 -2239.497,E2 -2239.497} C_VEL
LIN {X 0,Y 573.345,Z 589.544,A -85,B 0,C 180,E1 -2240.297,E2 -2240.297} C_VEL
LIN {X 0,Y 573.241,Z 599.115,A -85,B 0,C 180,E1 -2241.185,E2 -2241.185} C_VEL
LIN {X 0,Y 573.161,Z 606.962,A -85,B 0,C 180,E1 -2242.071,E2 -2242.071} C_VEL
LIN {X 0,Y 573.072,Z 614.955,A -85,B 0,C 180,E1 -2243.186,E2 -2243.186} C_VEL
LIN {X 0,Y 573.07,Z 621.681,A -85,B 0,C 180,E1 -2244.37,E2 -2244.37} C_VEL
LIN {X 0,Y 573.029,Z 626.372,A -85,B 0,C 180,E1 -2245.428,E2 -2245.428} C_VEL
LIN {X 0,Y 573.022,Z 629.957,A -85,B 0,C 180,E1 -2246.484,E2 -2246.484} C_VEL
LIN {X 0,Y 572.959,Z 631.808,A -85,B 0,C 180,E1 -2247.188,E2 -2247.188} C_VEL
LIN {X 0,Y 572.938,Z 633.198,A -85,B 0,C 180,E1 -2247.891,E2 -2247.891} C_VEL
LIN {X 0,Y 572.941,Z 634.785,A -85,B 0,C 180,E1 -2249.297,E2 -2249.297} C_VEL
LIN {X 0,Y 572.938,Z 635,A -85,B 0,C 180,E1 -2250,E2 -2250} C_VEL
LIN {X 0,Y 572.946,Z 634.186,A -85,B 0,C 180,E1 -2251.406,E2 -2251.406} C_VEL
LIN {X 0,Y 572.938,Z 633.2,A -85,B 0,C 180,E1 -2252.109,E2 -2252.109} C_VEL
LIN {X 0,Y 572.959,Z 631.81,A -85,B 0,C 180,E1 -2252.812,E2 -2252.812} C_VEL
LIN {X 0,Y 573.014,Z 628.896,A -85,B 0,C 180,E1 -2253.868,E2 -2253.868} C_VEL
LIN {X 0,Y 572.963,Z 624.949,A -85,B 0,C 180,E1 -2254.925,E2 -2254.925} C_VEL
LIN {X 0,Y 573.064,Z 618.878,A -85,B 0,C 180,E1 -2256.16,E2 -2256.16} C_VEL
LIN {X 0,Y 573.119,Z 612.239,A -85,B 0,C 180,E1 -2257.221,E2 -2257.221} C_VEL
LIN {X 0,Y 573.201,Z 603.992,A -85,B 0,C 180,E1 -2258.283,E2 -2258.283} C_VEL
LIN {X 0,Y 573.286,Z 595.541,A -85,B 0,C 180,E1 -2259.17,E2 -2259.17} C_VEL
LIN {X 0,Y 573.423,Z 585.101,A -85,B 0,C 180,E1 -2260.058,E2 -2260.058} C_VEL
LIN {X 0,Y 573.528,Z 573.358,A -85,B 0,C 180,E1 -2260.858,E2 -2260.858} C_VEL
LIN {X 0,Y 573.652,Z 562.288,A -85,B 0,C 180,E1 -2261.447,E2 -2261.447} C_VEL
LIN {X 0,Y 573.745,Z 549.18,A -85,B 0,C 180,E1 -2261.974,E2 -2261.974} C_VEL
LIN {X 0,Y 573.841,Z 536.531,A -85,B 0,C 180,E1 -2262.331,E2 -2262.331} C_VEL
LIN {X 0,Y 573.922,Z 523.333,A -85,B 0,C 180,E1 -2262.554,E2 -2262.554} C_VEL
LIN {X 0,Y 573.984,Z 426.422,A -85,B 0,C 180,E1 -2263.772,E2 -2263.772} C_VEL
LIN {X 0,Y 573.418,Z 422.441,A -85,B 0,C 180,E1 -2263.85,E2 -2263.85} C_VEL
LIN {X 0,Y 573.622,Z 399.373,A -85,B 0,C 180,E1 -2267.004,E2 -2267.004} C_VEL
LIN {X 0,Y 573.869,Z 377.402,A -85,B 0,C 180,E1 -2270.054,E2 -2270.054} C_VEL
LIN {X 0,Y 574.13,Z 356.07,A -85,B 0,C 180,E1 -2273.061,E2 -2273.061} C_VEL
LIN {X 0,Y 573.576,Z 351.686,A -85,B 0,C 180,E1 -2273.697,E2 -2273.697} C_VEL
LIN {X 0,Y 573.265,Z 350.081,A -85,B 0,C 180,E1 -2273.959,E2 -2273.959} C_VEL
LIN {X 0,Y 573.252,Z 350.074,A -85,B 0,C 180,E1 -2276.975,E2 -2276.975} C_VEL
LIN {X 0,Y 573.253,Z 350.075,A -85,B 0,C 180,E1 -2279.489,E2 -2279.489} C_VEL
LIN {X 0,Y 573.255,Z 350.08,A -85,B 0,C 180,E1 -2282.228,E2 -2282.228} C_VEL
LIN {X 0,Y 573.252,Z 350.074,A -85,B 0,C 180,E1 -2284.773,E2 -2284.773} C_VEL
LIN {X 0,Y 573.252,Z 350.073,A -85,B 0,C 180,E1 -2287.166,E2 -2287.166} C_VEL
LIN {X 0,Y 573.248,Z 350.077,A -85,B 0,C 180,E1 -2289.606,E2 -2289.606} C_VEL
LIN {X 0,Y 573.239,Z 350.075,A -85,B 0,C 180,E1 -2292.641,E2 -2292.641} C_VEL
LIN {X 0,Y 573.235,Z 350.081,A -85,B 0,C 180,E1 -2295.666,E2 -2295.666} C_VEL
LIN {X 0,Y 573.242,Z 350.075,A -85,B 0,C 180,E1 -2298.544,E2 -2298.544} C_VEL
LIN {X 0,Y 573.244,Z 350.076,A -85,B 0,C 180,E1 -2301.298,E2 -2301.298} C_VEL
LIN {X 0,Y 573.258,Z 350.079,A -85,B 0,C 180,E1 -2304.011,E2 -2304.011} C_VEL
